AssertResults.ReportResult(ExpectedSize := SIZEOF(Expected),
                           ExpectedTypeClass := IBaseLibrary.TypeClass.TYPE_BYTE,
                           ExpectedValue := ADR(Expected),
                           ActualSize := SIZEOF(Actual),
                           ActualTypeClass := IBaseLibrary.TypeClass.TYPE_BYTE,
                           ActualValue := ADR(Actual),
                           Message := Message,
                           TestInstancePath := TestInstancePath,
                           AlreadyReported => AlreadyReported);

IF NOT AlreadyReported AND Expected <> Actual THEN
    SetTestFailed(AssertionType := E_AssertionType.Type_BYTE,
                  AssertionMessage := Message);

    AssertMessageFormatter.LogAssertFailure(Expected := CONCAT(
                                                       STR1 := '0x',
                                                       STR2 := BYTE_TO_HEXSTR(in := Expected,
                                                                                            iPrecision := 2,
                                                                                            bLoCase := FALSE)),
                                            Actual := CONCAT(
                                                       STR1 := '0x',
                                                       STR2 := BYTE_TO_HEXSTR(in := Actual,
                                                                                            iPrecision := 2,
                                                                                            bLoCase := FALSE)),
                                            Message := Message,
                                            TestInstancePath := TestInstancePath);
END_IF
END_METHOD

// Asserts that two DATEs are equal. If they are not, an assertion error is created.
METHOD PUBLIC AssertEquals_DATE
VAR_INPUT
    Expected : DATE; // DATE expected value
    Actual : DATE; // DATE actual value
    Message : T_MaxString; // The identifying message for the assertion error
END_VAR
VAR
    TestInstancePath : T_MaxString;
    AlreadyReported : BOOL;
END_VAR
IF GVL_TcUnit.IgnoreCurrentTest OR GVL_TcUnit.CurrentTestIsFinished THEN
    RETURN;
END_IF

TestInstancePath := AddTestNameToInstancePath(TestInstancePath := FindTestSuiteInstancePath());

AssertResults.ReportResult(ExpectedSize := SIZEOF(Expected),
                           ExpectedTypeClass := IBaseLibrary.TypeClass.TYPE_DATE,
                           ExpectedValue := ADR(Expected),
                           ActualSize := SIZEOF(Actual),
                           ActualTypeClass := IBaseLibrary.TypeClass.TYPE_DATE,
                           ActualValue := ADR(Actual),
                           Message := Message,
                           TestInstancePath := TestInstancePath,
                           AlreadyReported => AlreadyReported);

IF NOT AlreadyReported AND Expected <> Actual THEN
    SetTestFailed(AssertionType := E_AssertionType.Type_DATE,
                  AssertionMessage := Message);

    AssertMessageFormatter.LogAssertFailure(Expected := DATE_TO_STRING(Expected),
                                            Actual := DATE_TO_STRING(Actual),
                                            Message := Message,
                                            TestInstancePath := TestInstancePath);
END_IF
END_METHOD

// Asserts that two DATE_AND_TIMEs are equal. If they are not, an assertion error is created.
METHOD PUBLIC AssertEquals_DATE_AND_TIME
VAR_INPUT
    Expected : DATE_AND_TIME; // DATE_AND_TIME expected value
    Actual : DATE_AND_TIME; // DATE_AND_TIME actual value
    Message : T_MaxString; // The identifying message for the assertion error
END_VAR
VAR
    TestInstancePath : T_MaxString;
    AlreadyReported : BOOL;
END_VAR
IF GVL_TcUnit.IgnoreCurrentTest OR GVL_TcUnit.CurrentTestIsFinished THEN
    RETURN;
END_IF

TestInstancePath := AddTestNameToInstancePath(TestInstancePath := FindTestSuiteInstancePath());

AssertResults.ReportResult(ExpectedSize := SIZEOF(Expected),
                           ExpectedTypeClass := IBaseLibrary.TypeClass.TYPE_DATEANDTIME,
                           ExpectedValue := ADR(Expected),
                           ActualSize := SIZEOF(Actual),
                           ActualTypeClass := IBaseLibrary.TypeClass.TYPE_DATEANDTIME,
                           ActualValue := ADR(Actual),
                           Message := Message,
                           TestInstancePath := TestInstancePath,
                           AlreadyReported => AlreadyReported);

IF NOT AlreadyReported AND Expected <> Actual THEN
    SetTestFailed(AssertionType := E_AssertionType.Type_DATE_AND_TIME,
                  AssertionMessage := Message);

    AssertMessageFormatter.LogAssertFailure(Expected := DT_TO_STRING(Expected),
                                            Actual := DT_TO_STRING(Actual),
                                            Message := Message,
                                            TestInstancePath := TestInstancePath);
END_IF
END_METHOD

// Asserts that two DINTs are equal. If they are not, an assertion error is created.
METHOD PUBLIC AssertEquals_DINT
VAR_INPUT
    Expected : DINT; // DINT expected value
    Actual : DINT; // DINT actual value
    Message : T_MaxString; // The identifying message for the assertion error
END_VAR
VAR
    TestInstancePath : T_MaxString;
    AlreadyReported : BOOL;
END_VAR
IF GVL_TcUnit.IgnoreCurrentTest OR GVL_TcUnit.CurrentTestIsFinished THEN
    RETURN;
END_IF

TestInstancePath := AddTestNameToInstancePath(TestInstancePath := FindTestSuiteInstancePath());

AssertResults.ReportResult(ExpectedSize := SIZEOF(Expected),
                           ExpectedTypeClass := IBaseLibrary.TypeClass.TYPE_DINT,
                           ExpectedValue := ADR(Expected),
                           ActualSize := SIZEOF(Actual),
                           ActualTypeClass := IBaseLibrary.TypeClass.TYPE_DINT,
                           ActualValue := ADR(Actual),
                           Message := Message,
                           TestInstancePath := TestInstancePath,
                           AlreadyReported => AlreadyReported);

IF NOT AlreadyReported AND Expected <> Actual THEN
    SetTestFailed(AssertionType := E_AssertionType.Type_DINT,
                  AssertionMessage := Message);

    AssertMessageFormatter.LogAssertFailure(Expected := DINT_TO_STRING(Expected),
                                            Actual := DINT_TO_STRING(Actual),
                                            Message := Message,
                                            TestInstancePath := TestInstancePath);
END_IF
END_METHOD

// Asserts that two DWORDs are equal. If they are not, an assertion error is created.
METHOD PUBLIC AssertEquals_DWORD
VAR_INPUT
    Expected : DWORD; // DWORD expected value
    Actual : DWORD; // DWORD actual value
    Message : T_MaxString; // The identifying message for the assertion error
END_VAR
VAR
    TestInstancePath : T_MaxString;
    AlreadyReported : BOOL;
END_VAR
IF GVL_TcUnit.IgnoreCurrentTest OR GVL_TcUnit.CurrentTestIsFinished THEN
    RETURN;
END_IF

TestInstancePath := AddTestNameToInstancePath(TestInstancePath := FindTestSuiteInstancePath());

AssertResults.ReportResult(ExpectedSize := SIZEOF(Expected),
                           ExpectedTypeClass := IBaseLibrary.TypeClass.TYPE_DWORD,
                           ExpectedValue := ADR(Expected),
                           ActualSize := SIZEOF(Actual),
                           ActualTypeClass := IBaseLibrary.TypeClass.TYPE_DWORD,
                           ActualValue := ADR(Actual),
                           Message := Message,
                           TestInstancePath := TestInstancePath,
                           AlreadyReported => AlreadyReported);

IF NOT AlreadyReported AND Expected <> Actual THEN
    SetTestFailed(AssertionType := E_AssertionType.Type_DWORD,
                  AssertionMessage := Message);

    AssertMessageFormatter.LogAssertFailure(Expected := CONCAT(
                                                            STR1 := '0x',
                                                            STR2 := DWORD_TO_HEXSTR(in := Expected,
                                                                                                  iPrecision := 8,
                                                                                                  bLoCase := FALSE)),
                                            Actual := CONCAT(
                                                           STR1 := '0x',
                                                           STR2 := DWORD_TO_HEXSTR(in := Actual,
                                                                                                 iPrecision := 8,
                                                                                                 bLoCase := FALSE)),
                                            Message := Message,
                                            TestInstancePath := TestInstancePath);
END_IF
END_METHOD

// Asserts that two INTs are equal. If they are not, an assertion error is created.
METHOD PUBLIC AssertEquals_INT
VAR_INPUT
    Expected : INT; // INT expected value
    Actual : INT; // INT actual value
    Message : T_MaxString; // The identifying message for the assertion error
END_VAR
VAR
    TestInstancePath : T_MaxString;
    AlreadyReported : BOOL;
END_VAR
IF GVL_TcUnit.IgnoreCurrentTest OR GVL_TcUnit.CurrentTestIsFinished THEN
    RETURN;
END_IF

TestInstancePath := AddTestNameToInstancePath(TestInstancePath := FindTestSuiteInstancePath());

AssertResults.ReportResult(ExpectedSize := SIZEOF(Expected),
                           ExpectedTypeClass := IBaseLibrary.TypeClass.TYPE_INT,
                           ExpectedValue := ADR(Expected),
                           ActualSize := SIZEOF(Actual),
                           ActualTypeClass := IBaseLibrary.TypeClass.TYPE_INT,
                           ActualValue := ADR(Actual),
                           Message := Message,
                           TestInstancePath := TestInstancePath,
                           AlreadyReported => AlreadyReported);

IF NOT AlreadyReported AND Expected <> Actual THEN
    SetTestFailed(AssertionType := E_AssertionType.Type_INT,
                  AssertionMessage := Message);

    AssertMessageFormatter.LogAssertFailure(Expected := INT_TO_STRING(Expected),
                                            Actual := INT_TO_STRING(Actual),
                                            Message := Message,
                                            TestInstancePath := TestInstancePath);
END_IF
END_METHOD

// Asserts that two LINTs are equal. If they are not, an assertion error is created.
METHOD PUBLIC AssertEquals_LINT
VAR_INPUT
    Expected : LINT; // LINT expected value
    Actual : LINT; // LINT actual value
    Message : T_MaxString; // The identifying message for the assertion error
END_VAR
VAR
    TestInstancePath : T_MaxString;
    AlreadyReported : BOOL;
END_VAR
IF GVL_TcUnit.IgnoreCurrentTest OR GVL_TcUnit.CurrentTestIsFinished THEN
    RETURN;
END_IF

TestInstancePath := AddTestNameToInstancePath(TestInstancePath := FindTestSuiteInstancePath());

AssertResults.ReportResult(ExpectedSize := SIZEOF(Expected),
                           ExpectedTypeClass := IBaseLibrary.TypeClass.TYPE_LINT,
                           ExpectedValue := ADR(Expected),
                           ActualSize := SIZEOF(Actual),
                           ActualTypeClass := IBaseLibrary.TypeClass.TYPE_LINT,
                           ActualValue := ADR(Actual),
                           Message := Message,
                           TestInstancePath := TestInstancePath,
                           AlreadyReported => AlreadyReported);

IF NOT AlreadyReported AND Expected <> Actual THEN
    SetTestFailed(AssertionType := E_AssertionType.Type_LINT,
                  AssertionMessage := Message);

    AssertMessageFormatter.LogAssertFailure(Expected := LINT_TO_STRING(Expected),
                                            Actual := LINT_TO_STRING(Actual),
                                            Message := Message,
                                            TestInstancePath := TestInstancePath);
END_IF
END_METHOD

// Asserts that two LREALs are equal to within a positive delta. If they are not, an assertion error is created.
METHOD PUBLIC AssertEquals_LREAL
VAR_INPUT
    Expected : LREAL; // LREAL expected value
    Actual : LREAL; // LREAL actual value
    Delta : LREAL; // The maximum delta between the absolute value of expected and actual for which both numbers are still considered equal
    Message : T_MaxString; // The identifying message for the assertion error
END_VAR
VAR
    Equals : BOOL := TRUE;
    TestInstancePath : T_MaxString;
    AlreadyReported : BOOL;
END_VAR
IF GVL_TcUnit.IgnoreCurrentTest OR GVL_TcUnit.CurrentTestIsFinished THEN
    RETURN;
END_IF

TestInstancePath := AddTestNameToInstancePath(TestInstancePath := FindTestSuiteInstancePath());

AssertResults.ReportResult(ExpectedSize := SIZEOF(Expected),
                           ExpectedTypeClass := IBaseLibrary.TypeClass.TYPE_LREAL,
                           ExpectedValue := ADR(Expected),
                           ActualSize := SIZEOF(Actual),
                           ActualTypeClass := IBaseLibrary.TypeClass.TYPE_LREAL,
                           ActualValue := ADR(Actual),
                           Message := Message,
                           TestInstancePath := TestInstancePath,
                           AlreadyReported => AlreadyReported);

IF NOT AlreadyReported THEN
    IF LrealIsNaN (Delta) THEN
        Equals := FALSE;
        Message := CONCAT(STR1 := Message, STR2 := ', value of delta is NaN.');
    ELSIF (LrealIsNaN (Expected)
    OR     LrealIsNaN (Actual)) THEN
        Equals := FALSE;
        Message := CONCAT(STR1 := Message, STR2 := ', value of Expected or Actual is NaN.');
    ELSIF ABS(Expected - Actual) > Delta THEN
        Equals := FALSE;
    END_IF

    IF NOT Equals THEN
        SetTestFailed(AssertionType := E_AssertionType.Type_LREAL,
                      AssertionMessage := Message);

        AssertMessageFormatter.LogAssertFailure(Expected := LREAL_TO_STRING(Expected),
                                                Actual := LREAL_TO_STRING(Actual),
                                                Message := Message,
                                                TestInstancePath := TestInstancePath);
    END_IF
END_IF
END_METHOD

// Asserts that two LTIMEs are equal. If they are not, an assertion error is created.
METHOD PUBLIC AssertEquals_LTIME
VAR_INPUT
    Expected : LTIME; // LTIME expected value
    Actual : LTIME; // LTIME actual value
    Message : T_MaxString; // The identifying message for the assertion error
END_VAR
VAR
    TestInstancePath : T_MaxString;
    AlreadyReported : BOOL;
END_VAR
IF GVL_TcUnit.IgnoreCurrentTest OR GVL_TcUnit.CurrentTestIsFinished THEN
    RETURN;
END_IF

TestInstancePath := AddTestNameToInstancePath(TestInstancePath := FindTestSuiteInstancePath());

AssertResults.ReportResult(ExpectedSize := SIZEOF(Expected),
                           ExpectedTypeClass := IBaseLibrary.TypeClass.TYPE_LTIME,
                           ExpectedValue := ADR(Expected),
                           ActualSize := SIZEOF(Actual),
                           ActualTypeClass := IBaseLibrary.TypeClass.TYPE_LTIME,
                           ActualValue := ADR(Actual),
                           Message := Message,
                           TestInstancePath := TestInstancePath,
                           AlreadyReported => AlreadyReported);

IF NOT AlreadyReported AND Expected <> Actual THEN
    SetTestFailed(AssertionType := E_AssertionType.Type_LTIME,
                  AssertionMessage := Message);

    AssertMessageFormatter.LogAssertFailure(Expected := LTIME_TO_STRING(Expected),
                                            Actual := LTIME_TO_STRING(Actual),
                                            Message := Message,
                                            TestInstancePath := TestInstancePath);
END_IF
END_METHOD

// Asserts that two LWORDs are equal. If they are not, an assertion error is created.
METHOD PUBLIC AssertEquals_LWORD
VAR_INPUT
    Expected : LWORD; // LWORD expected value
    Actual : LWORD; // LWORD actual value
    Message : T_MaxString; // The identifying message for the assertion error
END_VAR
VAR
    TestInstancePath : T_MaxString;
    AlreadyReported : BOOL;
END_VAR
IF GVL_TcUnit.IgnoreCurrentTest OR GVL_TcUnit.CurrentTestIsFinished THEN
    RETURN;
END_IF

TestInstancePath := AddTestNameToInstancePath(TestInstancePath := FindTestSuiteInstancePath());

AssertResults.ReportResult(ExpectedSize := SIZEOF(Expected),
                           ExpectedTypeClass := IBaseLibrary.TypeClass.TYPE_LWORD,
                           ExpectedValue := ADR(Expected),
                           ActualSize := SIZEOF(Actual),
                           ActualTypeClass := IBaseLibrary.TypeClass.TYPE_LWORD,
                           ActualValue := ADR(Actual),
                           Message := Message,
                           TestInstancePath := TestInstancePath,
                           AlreadyReported => AlreadyReported);

IF NOT AlreadyReported AND Expected <> Actual THEN
    SetTestFailed(AssertionType := E_AssertionType.Type_LWORD,
                  AssertionMessage := Message);

    AssertMessageFormatter.LogAssertFailure(Expected := CONCAT(
                                                            STR1 := '0x',
                                                            STR2 := LWORD_TO_HEXSTR(in := Expected,
                                                                                                  iPrecision := 16,
                                                                                                  bLoCase := FALSE)),
                                            Actual := CONCAT(
                                                            STR1 := '0x',
                                                            STR2 := LWORD_TO_HEXSTR(in := Actual,
                                                                                                  iPrecision := 16,
                                                                                                  bLoCase := FALSE)),
                                            Message := Message,
                                            TestInstancePath := TestInstancePath);
END_IF
END_METHOD

// Asserts that two REALs are equal to within a positive delta. If they are not, an assertion error is created.
METHOD PUBLIC AssertEquals_REAL
VAR_INPUT
    Expected : REAL; // REAL expected value
    Actual : REAL; // REAL actual value
    Delta : REAL;  // The maximum delta between the absolute value of expected and actual for which both numbers are still considered equal
    Message : T_MaxString; // The identifying message for the assertion error
END_VAR
VAR
    Equals : BOOL := TRUE;
    TestInstancePath : T_MaxString;
    AlreadyReported : BOOL;
END_VAR
IF GVL_TcUnit.IgnoreCurrentTest OR GVL_TcUnit.CurrentTestIsFinished THEN
    RETURN;
END_IF

TestInstancePath := AddTestNameToInstancePath(TestInstancePath := FindTestSuiteInstancePath());

AssertResults.ReportResult(ExpectedSize := SIZEOF(Expected),
                           ExpectedTypeClass := IBaseLibrary.TypeClass.TYPE_REAL,
                           ExpectedValue := ADR(Expected),
                           ActualSize := SIZEOF(Actual),
                           ActualTypeClass := IBaseLibrary.TypeClass.TYPE_REAL,
                           ActualValue := ADR(Actual),
                           Message := Message,
                           TestInstancePath := TestInstancePath,
                           AlreadyReported => AlreadyReported);

IF NOT AlreadyReported THEN
    IF RealIsNaN (Delta) THEN
        Equals := FALSE;
        Message := CONCAT(STR1 := Message, STR2 := ', value of delta is NaN.');
    ELSIF (RealIsNaN (Expected)
    OR     RealIsNaN (Actual)) THEN
        Equals := FALSE;
        Message := CONCAT(STR1 := Message, STR2 := ', value of Expected or Actual is NaN.');
    ELSIF ABS(Expected - Actual) > Delta THEN
        Equals := FALSE;
    END_IF

    IF NOT Equals THEN
        SetTestFailed(AssertionType := E_AssertionType.Type_REAL,
                      AssertionMessage := Message);

        AssertMessageFormatter.LogAssertFailure(Expected := REAL_TO_STRING(Expected),
                                                Actual := REAL_TO_STRING(Actual),
                                                Message := Message,
                                                TestInstancePath := TestInstancePath);
    END_IF
END_IF
END_METHOD

// Asserts that two SINTs are equal. If they are not, an assertion error is created.
METHOD PUBLIC AssertEquals_SINT
VAR_INPUT
    Expected : SINT; // SINT expected value
    Actual : SINT; // SINT actual value
    Message : T_MaxString; // The identifying message for the assertion error
END_VAR
VAR
    TestInstancePath : T_MaxString;
    AlreadyReported : BOOL;
END_VAR
IF GVL_TcUnit.IgnoreCurrentTest OR GVL_TcUnit.CurrentTestIsFinished THEN
    RETURN;
END_IF

TestInstancePath := AddTestNameToInstancePath(TestInstancePath := FindTestSuiteInstancePath());

AssertResults.ReportResult(ExpectedSize := SIZEOF(Expected),
                           ExpectedTypeClass := IBaseLibrary.TypeClass.TYPE_SINT,
                           ExpectedValue := ADR(Expected),
                           ActualSize := SIZEOF(Actual),
                           ActualTypeClass := IBaseLibrary.TypeClass.TYPE_SINT,
                           ActualValue := ADR(Actual),
                           Message := Message,
                           TestInstancePath := TestInstancePath,
                           AlreadyReported => AlreadyReported);

IF NOT AlreadyReported AND Expected <> Actual THEN
    SetTestFailed(AssertionType := E_AssertionType.Type_SINT,
                  AssertionMessage := Message);

    AssertMessageFormatter.LogAssertFailure(Expected := SINT_TO_STRING(Expected),
                                            Actual := SINT_TO_STRING(Actual),
                                            Message := Message,
                                            TestInstancePath := TestInstancePath);
END_IF
END_METHOD

// Asserts that two STRINGs are equal. If they are not, an assertion error is created.
METHOD PUBLIC AssertEquals_STRING
VAR_INPUT
    Expected : T_MaxString; // STRING expected value
    Actual : T_MaxString; // STRING actual value
    Message : T_MaxString; // The identifying message for the assertion error
END_VAR
VAR
    TestInstancePath : T_MaxString;
    AlreadyReported : BOOL;
END_VAR
IF GVL_TcUnit.IgnoreCurrentTest OR GVL_TcUnit.CurrentTestIsFinished THEN
    RETURN;
END_IF

TestInstancePath := AddTestNameToInstancePath(TestInstancePath := FindTestSuiteInstancePath());

AssertResults.ReportResult(ExpectedSize := SIZEOF(Expected),
                           ExpectedTypeClass := IBaseLibrary.TypeClass.TYPE_STRING,
                           ExpectedValue := ADR(Expected),
                           ActualSize := SIZEOF(Actual),
                           ActualTypeClass := IBaseLibrary.TypeClass.TYPE_STRING,
                           ActualValue := ADR(Actual),
                           Message := Message,
                           TestInstancePath := TestInstancePath,
                           AlreadyReported => AlreadyReported);

IF NOT AlreadyReported AND (LEN(STR := Expected) <> LEN(STR := Actual) OR (Expected <> Actual)) THEN
    SetTestFailed(AssertionType := E_AssertionType.Type_STRING,
                  AssertionMessage := Message);

    AssertMessageFormatter.LogAssertFailure(Expected := Expected,
                                            Actual := Actual,
                                            Message := Message,
                                            TestInstancePath := TestInstancePath);
END_IF
END_METHOD

// Asserts that two TIMEs are equal. If they are not, an assertion error is created.
METHOD PUBLIC AssertEquals_TIME
VAR_INPUT
    Expected : TIME; // TIME expected value
    Actual : TIME; // TIME actual value
    Message : T_MaxString; // The identifying message for the assertion error
END_VAR
VAR
    TestInstancePath : T_MaxString;
    AlreadyReported : BOOL;
END_VAR
IF GVL_TcUnit.IgnoreCurrentTest OR GVL_TcUnit.CurrentTestIsFinished THEN
    RETURN;
END_IF

TestInstancePath := AddTestNameToInstancePath(TestInstancePath := FindTestSuiteInstancePath());

AssertResults.ReportResult(ExpectedSize := SIZEOF(Expected),
                           ExpectedTypeClass := IBaseLibrary.TypeClass.TYPE_TIME,
                           ExpectedValue := ADR(Expected),
                           ActualSize := SIZEOF(Actual),
                           ActualTypeClass := IBaseLibrary.TypeClass.TYPE_TIME,
                           ActualValue := ADR(Actual),
                           Message := Message,
                           TestInstancePath := TestInstancePath,
                           AlreadyReported => AlreadyReported);

IF NOT AlreadyReported AND Expected <> Actual THEN
    SetTestFailed(AssertionType := E_AssertionType.Type_TIME,
                  AssertionMessage := Message);

    AssertMessageFormatter.LogAssertFailure(Expected := TIME_TO_STRING(Expected),
                                            Actual := TIME_TO_STRING(Actual),
                                            Message := Message,
                                            TestInstancePath := TestInstancePath);
END_IF
END_METHOD

// Asserts that two TIME_OF_DAYs are equal. If they are not, an assertion error is created.
METHOD PUBLIC AssertEquals_TIME_OF_DAY
VAR_INPUT
    Expected : TIME_OF_DAY; // TIME_OF_DAY expected value
    Actual : TIME_OF_DAY; // TIME_OF_DAY actual value
    Message : T_MaxString; // The identifying message for the assertion error
END_VAR
VAR
    TestInstancePath : T_MaxString;
    AlreadyReported : BOOL;
END_VAR
IF GVL_TcUnit.IgnoreCurrentTest OR GVL_TcUnit.CurrentTestIsFinished THEN
    RETURN;
END_IF

TestInstancePath := AddTestNameToInstancePath(TestInstancePath := FindTestSuiteInstancePath());

AssertResults.ReportResult(ExpectedSize := SIZEOF(Expected),
                           ExpectedTypeClass := IBaseLibrary.TypeClass.TYPE_TIMEOFDAY,
                           ExpectedValue := ADR(Expected),
                           ActualSize := SIZEOF(Actual),
                           ActualTypeClass := IBaseLibrary.TypeClass.TYPE_TIMEOFDAY,
                           ActualValue := ADR(Actual),
                           Message := Message,
                           TestInstancePath := TestInstancePath,
                           AlreadyReported => AlreadyReported);

IF NOT AlreadyReported AND Expected <> Actual THEN
    SetTestFailed(AssertionType := E_AssertionType.Type_TIME_OF_DAY,
                  AssertionMessage := Message);

    AssertMessageFormatter.LogAssertFailure(Expected := TOD_TO_STRING(Expected),
                                            Actual := TOD_TO_STRING(Actual),
                                            Message := Message,
                                            TestInstancePath := TestInstancePath);
END_IF
END_METHOD

// Asserts that two UDINTs are equal. If they are not, an assertion error is created.
METHOD PUBLIC AssertEquals_UDINT
VAR_INPUT
    Expected : UDINT; // UDINT expected value
    Actual : UDINT; // UDINT actual value
    Message : T_MaxString; // The identifying message for the assertion error
END_VAR
VAR
    TestInstancePath : T_MaxString;
    AlreadyReported : BOOL;
END_VAR
IF GVL_TcUnit.IgnoreCurrentTest OR GVL_TcUnit.CurrentTestIsFinished THEN
    RETURN;
END_IF

TestInstancePath := AddTestNameToInstancePath(TestInstancePath := FindTestSuiteInstancePath());

AssertResults.ReportResult(ExpectedSize := SIZEOF(Expected),
                           ExpectedTypeClass := IBaseLibrary.TypeClass.TYPE_UDINT,
                           ExpectedValue := ADR(Expected),
                           ActualSize := SIZEOF(Actual),
                           ActualTypeClass := IBaseLibrary.TypeClass.TYPE_UDINT,
                           ActualValue := ADR(Actual),
                           Message := Message,
                           TestInstancePath := TestInstancePath,
                           AlreadyReported => AlreadyReported);

IF NOT AlreadyReported AND Expected <> Actual THEN
    SetTestFailed(AssertionType := E_AssertionType.Type_UDINT,
                  AssertionMessage := Message);

    AssertMessageFormatter.LogAssertFailure(Expected := UDINT_TO_STRING(Expected),
                                            Actual := UDINT_TO_STRING(Actual),
                                            Message := Message,
                                            TestInstancePath := TestInstancePath);
END_IF
END_METHOD

// Asserts that two UINTs are equal. If they are not, an assertion error is created.
METHOD PUBLIC AssertEquals_UINT
VAR_INPUT
    Expected : UINT; // UINT expected value
    Actual : UINT; // UINT actual value
    Message : T_MaxString; // The identifying message for the assertion error
END_VAR
VAR
    TestInstancePath : T_MaxString;
    AlreadyReported : BOOL;
END_VAR
IF GVL_TcUnit.IgnoreCurrentTest OR GVL_TcUnit.CurrentTestIsFinished THEN
    RETURN;
END_IF

TestInstancePath := AddTestNameToInstancePath(TestInstancePath := FindTestSuiteInstancePath());

AssertResults.ReportResult(ExpectedSize := SIZEOF(Expected),
                           ExpectedTypeClass := IBaseLibrary.TypeClass.TYPE_UINT,
                           ExpectedValue := ADR(Expected),
                           ActualSize := SIZEOF(Actual),
                           ActualTypeClass := IBaseLibrary.TypeClass.TYPE_UINT,
                           ActualValue := ADR(Actual),
                           Message := Message,
                           TestInstancePath := TestInstancePath,
                           AlreadyReported => AlreadyReported);

IF NOT AlreadyReported AND Expected <> Actual THEN
    SetTestFailed(AssertionType := E_AssertionType.Type_UINT,
                  AssertionMessage := Message);

    AssertMessageFormatter.LogAssertFailure(Expected := UINT_TO_STRING(Expected),
                                            Actual := UINT_TO_STRING(Actual),
                                            Message := Message,
                                            TestInstancePath := TestInstancePath);
END_IF
END_METHOD

// Asserts that two ULINTs are equal. If they are not, an assertion error is created.
METHOD PUBLIC AssertEquals_ULINT
VAR_INPUT
    Expected : ULINT; // ULINT expected value
    Actual : ULINT; // ULINT actual value
    Message : T_MaxString; // The identifying message for the assertion error
END_VAR
VAR
    TestInstancePath : T_MaxString;
    AlreadyReported : BOOL;
END_VAR
IF GVL_TcUnit.IgnoreCurrentTest OR GVL_TcUnit.CurrentTestIsFinished THEN
    RETURN;
END_IF

TestInstancePath := AddTestNameToInstancePath(TestInstancePath := FindTestSuiteInstancePath());

AssertResults.ReportResult(ExpectedSize := SIZEOF(Expected),
                           ExpectedTypeClass := IBaseLibrary.TypeClass.TYPE_ULINT,
                           ExpectedValue := ADR(Expected),
                           ActualSize := SIZEOF(Actual),
                           ActualTypeClass := IBaseLibrary.TypeClass.TYPE_ULINT,
                           ActualValue := ADR(Actual),
                           Message := Message,
                           TestInstancePath := TestInstancePath,
                           AlreadyReported => AlreadyReported);

IF NOT AlreadyReported AND Expected <> Actual THEN
    SetTestFailed(AssertionType := E_AssertionType.Type_ULINT,
                  AssertionMessage := Message);

    AssertMessageFormatter.LogAssertFailure(Expected := ULINT_TO_STRING(Expected),
                                            Actual := ULINT_TO_STRING(Actual),
                                            Message := Message,
                                            TestInstancePath := TestInstancePath);
END_IF
END_METHOD

// Asserts that two USINTs are equal. If they are not, an assertion error is created.
METHOD PUBLIC AssertEquals_USINT
VAR_INPUT
    Expected : USINT; // USINT expected value
    Actual : USINT; // USINT actual value
    Message : T_MaxString; // The identifying message for the assertion error
END_VAR
VAR
    AlreadyReported : BOOL;
    TestInstancePath : T_MaxString;
END_VAR
IF GVL_TcUnit.IgnoreCurrentTest OR GVL_TcUnit.CurrentTestIsFinished THEN
    RETURN;
END_IF

TestInstancePath := AddTestNameToInstancePath(TestInstancePath := FindTestSuiteInstancePath());

AssertResults.ReportResult(ExpectedSize := SIZEOF(Expected),
                           ExpectedTypeClass := IBaseLibrary.TypeClass.TYPE_USINT,
                           ExpectedValue := ADR(Expected),
                           ActualSize := SIZEOF(Actual),
                           ActualTypeClass := IBaseLibrary.TypeClass.TYPE_USINT,
                           ActualValue := ADR(Actual),
                           Message := Message,
                           TestInstancePath := TestInstancePath,
                           AlreadyReported => AlreadyReported);

IF NOT AlreadyReported AND Expected <> Actual THEN
    SetTestFailed(AssertionType := E_AssertionType.Type_USINT,
                  AssertionMessage := Message);

    AssertMessageFormatter.LogAssertFailure(Expected := USINT_TO_STRING(Expected),
                                            Actual := USINT_TO_STRING(Actual),
                                            Message := Message,
                                            TestInstancePath := TestInstancePath);
END_IF
END_METHOD

// Asserts that two WORDs are equal. If they are not, an assertion error is created.
METHOD PUBLIC AssertEquals_WORD
VAR_INPUT
    Expected : WORD; // WORD expected value
    Actual : WORD; // WORD actual value
    Message : T_MaxString; // The identifying message for the assertion error
END_VAR
VAR
    TestInstancePath : T_MaxString;
    AlreadyReported : BOOL;
END_VAR
IF GVL_TcUnit.IgnoreCurrentTest OR GVL_TcUnit.CurrentTestIsFinished THEN
    RETURN;
END_IF

TestInstancePath := AddTestNameToInstancePath(TestInstancePath := FindTestSuiteInstancePath());

AssertResults.ReportResult(ExpectedSize := SIZEOF(Expected),
                           ExpectedTypeClass := IBaseLibrary.TypeClass.TYPE_WORD,
                           ExpectedValue := ADR(Expected),
                           ActualSize := SIZEOF(Actual),
                           ActualTypeClass := IBaseLibrary.TypeClass.TYPE_WORD,
                           ActualValue := ADR(Actual),
                           Message := Message,
                           TestInstancePath := TestInstancePath,
                           AlreadyReported => AlreadyReported);

IF NOT AlreadyReported AND Expected <> Actual THEN
    SetTestFailed(AssertionType := E_AssertionType.Type_WORD,
                  AssertionMessage := Message);

    AssertMessageFormatter.LogAssertFailure(Expected := CONCAT(
                                                            STR1 := '0x',
                                                            STR2 := WORD_TO_HEXSTR(in := Expected,
                                                                                                 iPrecision := 4,
                                                                                                 bLoCase := FALSE)),
                                            Actual := CONCAT(
                                                            STR1 := '0x',
                                                            STR2 := WORD_TO_HEXSTR(in := Actual,
                                                                                                 iPrecision := 4,
                                                                                                 bLoCase := FALSE)),
                                            Message := Message,
                                            TestInstancePath := TestInstancePath);
END_IF
END_METHOD

// Asserts that two WSTRINGs are equal. If they are not, an assertion error is created.
METHOD PUBLIC AssertEquals_WSTRING
VAR_INPUT
    Expected : WSTRING(255); // WSTRING expected value
    Actual : WSTRING(255); // WSTRING actual value
    Message : T_MaxString; // The identifying message for the assertion error
END_VAR
VAR
    TestInstancePath : T_MaxString;
    AlreadyReported : BOOL;
END_VAR
IF GVL_TcUnit.IgnoreCurrentTest OR GVL_TcUnit.CurrentTestIsFinished THEN
    RETURN;
END_IF

TestInstancePath := AddTestNameToInstancePath(TestInstancePath := FindTestSuiteInstancePath());

AssertResults.ReportResult(ExpectedSize := SIZEOF(Expected),
                           ExpectedTypeClass := IBaseLibrary.TypeClass.TYPE_WSTRING,
                           ExpectedValue := ADR(Expected),
                           ActualSize := SIZEOF(Actual),
                           ActualTypeClass := IBaseLibrary.TypeClass.TYPE_WSTRING,
                           ActualValue := ADR(Actual),
                           Message := Message,
                           TestInstancePath := TestInstancePath,
                           AlreadyReported => AlreadyReported);

IF NOT AlreadyReported AND (WLEN(STR := Expected) <> WLEN(STR := Actual) OR (Expected <> Actual)) THEN
    SetTestFailed(AssertionType := E_AssertionType.Type_WSTRING,
                  AssertionMessage := Message);

    AssertMessageFormatter.LogAssertFailure(Expected := 'Not possible to print EXP unicode WSTRING value',
                                            Actual := 'Not possible to print ACT unicode WSTRING value',
                                            Message := Message,
                                            TestInstancePath := TestInstancePath);
END_IF
END_METHOD

// Asserts that a condition is false. If it is not, an assertion error is created.
METHOD PUBLIC AssertFalse
VAR_INPUT
    Condition : BOOL; // Condition to be checked
    Message : T_MaxString; // The identifying message for the assertion error
END_VAR
AssertEquals_BOOL(Expected := FALSE,
                  Actual := Condition,
                  Message := Message);
END_METHOD

// Asserts that a condition is true. If it is not, an assertion error is created.
METHOD PUBLIC AssertTrue
VAR_INPUT
    Condition : BOOL; // Condition to be checked
    Message : T_MaxString; // The identifying message for the assertion error
END_VAR
AssertEquals_BOOL(Expected := TRUE,
                  Actual := Condition,
                  Message := Message);
END_METHOD

METHOD INTERNAL CalculateAndSetNumberOfAssertsForTest
VAR_INPUT
    TestName : T_MaxString;
END_VAR
VAR
    TestInstancePath : T_MaxString;
    TotalNumberOfAsserts : UINT;
    NumberOfAsserts : UINT;
    NumberOfArrayAsserts : UINT;
    
    IteratorCounter : UINT;
END_VAR
TestInstancePath := AddTestNameToInstancePath(FindTestSuiteInstancePath());
NumberOfAsserts := AssertResults.GetNumberOfAssertsForTest(CompleteTestInstancePath := TestInstancePath);
NumberOfArrayAsserts := AssertArrayResults.GetNumberOfArrayAssertsForTest(CompleteTestInstancePath := TestInstancePath);
TotalNumberOfAsserts := NumberOfAsserts + NumberOfArrayAsserts;

IF TotalNumberOfAsserts > 0 THEN
    IF NumberOfTests > 0 THEN
        FOR IteratorCounter := 1 TO NumberOfTests BY 1 DO
            IF Tests[IteratorCounter].GetName() = TestName THEN
                Tests[IteratorCounter].SetNumberOfAssertions(NoOfAssertions := TotalNumberOfAsserts);
                RETURN;
            END_IF
        END_FOR
    END_IF
END_IF
END_METHOD

METHOD INTERNAL CalculateDuration
VAR_INPUT
    FinishedAt : LWORD; // CPU cycle counter with 100ns precision
END_VAR
IF Duration = 0.0 THEN
	Duration := LWORD_TO_LREAL(FinishedAt - StartedAt) * GVL_TcUnit.HundredNanosecondToSecond; // Seconds
END_IF
END_METHOD

METHOD FB_init : BOOL
VAR_INPUT
    bInitRetains : BOOL; // if TRUE, the retain variables are initialized (warm start / cold start)
    bInCopyCode : BOOL;  // if TRUE, the instance afterwards gets moved into the copy code (online change)
END_VAR
GVL_TcUnit.NumberOfInitializedTestSuites := GVL_TcUnit.NumberOfInitializedTestSuites + 1;
GVL_TcUnit.TestSuiteAddresses[GVL_TcUnit.NumberOfInitializedTestSuites] := THIS;
END_METHOD

// Searches for the instance path of the calling function block
METHOD PRIVATE FindTestSuiteInstancePath : T_MaxString
FindTestSuiteInstancePath := GetInstancePath();
END_METHOD

METHOD INTERNAL GetDuration : LREAL
GetDuration := Duration;
END_METHOD

METHOD INTERNAL GetHasStartedRunning : BOOL
GetHasStartedRunning := StartedAt > 0;
END_METHOD

METHOD INTERNAL GetInstancePath : T_MaxString
GetInstancePath := InstancePath;
END_METHOD

METHOD INTERNAL GetNumberOfFailedTests : UINT
VAR
    Counter : UINT;
    FailedTestsCount : UINT;
    NumberOfTestsToAnalyse : UINT(1..GVL_Param_TcUnit.MaxNumberOfTestsForEachTestSuite);
    NumberOfTestOverArrayLimit : UINT;
END_VAR
// Limit the test analyse to the max array limit of 'Tests[]'
NumberOfTestsToAnalyse := GetNumberOfTestsToAnalyse();
IF GetNumberOfTests() > NumberOfTestsToAnalyse THEN
    NumberOfTestOverArrayLimit := GetNumberOfTests()-NumberOfTestsToAnalyse;
END_IF

FOR Counter := 1 TO NumberOfTestsToAnalyse BY 1 DO
    IF Tests[Counter].IsFailed() THEN
        FailedTestsCount := FailedTestsCount + 1;
    END_IF
END_FOR

GetNumberOfFailedTests := FailedTestsCount + NumberOfTestOverArrayLimit;
END_METHOD

METHOD INTERNAL GetNumberOfSkippedTests : UINT
VAR
    Counter : UINT;
    SkippedTestsCount : UINT;
    NumberOfTestsToAnalyse : UINT(1..GVL_Param_TcUnit.MaxNumberOfTestsForEachTestSuite);
END_VAR
// Limit the test analyse to the max array limit of 'Tests[]'
NumberOfTestsToAnalyse := GetNumberOfTestsToAnalyse();

FOR Counter := 1 TO NumberOfTestsToAnalyse BY 1 DO
    IF Tests[Counter].IsSkipped() THEN
        SkippedTestsCount := SkippedTestsCount + 1;
    END_IF
END_FOR

GetNumberOfSkippedTests := SkippedTestsCount;
END_METHOD

METHOD INTERNAL GetNumberOfSuccessfulTests : UINT
GetNumberOfSuccessfulTests := GetNumberOfTests() - GetNumberOfFailedTests() - GetNumberOfSkippedTests();
END_METHOD

METHOD INTERNAL GetNumberOfTests : UINT
GetNumberOfTests := NumberOfTests;
END_METHOD

METHOD INTERNAL GetNumberOfTestsToAnalyse : UINT
GetNumberOfTestsToAnalyse := MIN(GetNumberOfTests(), GVL_Param_TcUnit.MaxNumberOfTestsForEachTestSuite);
END_METHOD

METHOD GetTestByName : REFERENCE TO FB_Test
VAR_INPUT
  TestName : T_MaxString;
END_VAR
VAR
  IteratorCounter : UINT;
  NumberOfTestsToAnalyse : UINT(1..GVL_Param_TcUnit.MaxNumberOfTestSuites);
END_VAR
NumberOfTestsToAnalyse := GetNumberOfTestsToAnalyse();
FOR IteratorCounter := 1 TO NumberOfTestsToAnalyse BY 1 DO
  IF Tests[IteratorCounter].GetName() = TestName THEN
    GetTestByName REF= Tests[IteratorCounter];
    RETURN;
	END_IF
END_FOR
END_METHOD

// This method returns the test at the n'th position, ranging from 1.. NumberOfTests
METHOD INTERNAL GetTestByPosition : FB_Test
VAR_INPUT
    Position : UINT(1..GVL_Param_TcUnit.MaxNumberOfTestsForEachTestSuite);
END_VAR
GetTestByPosition := Tests[Position];
END_METHOD

METHOD INTERNAL GetTestOrderNumber : UINT(0..GVL_Param_TcUnit.MaxNumberOfTestsForEachTestSuite);
VAR_INPUT
    TestName : T_MaxString;
END_VAR
VAR
    IteratorCounter : UINT;
    NumberOfTestsToAnalyse : UINT(1..GVL_Param_TcUnit.MaxNumberOfTestsForEachTestSuite);
END_VAR
// Limit the test analyse to the max array limit of 'Tests[]'
NumberOfTestsToAnalyse := GetNumberOfTestsToAnalyse();

FOR IteratorCounter := 1 TO NumberOfTestsToAnalyse BY 1 DO
    IF Tests[IteratorCounter].GetName() = TestName THEN
        GetTestOrderNumber := Tests[IteratorCounter].GetTestOrder();
        RETURN;
    END_IF
END_FOR
END_METHOD

METHOD INTERNAL IsTestFinished : BOOL
VAR_INPUT
    TestName : T_MaxString;
END_VAR
VAR
    IteratorCounter : UINT;
    NumberOfTestsToAnalyse : UINT(0..GVL_Param_TcUnit.MaxNumberOfTestsForEachTestSuite);
END_VAR
// Limit the test analyse to the max array limit of 'Tests[]'
NumberOfTestsToAnalyse := GetNumberOfTestsToAnalyse();

IsTestFinished := FALSE;
FOR IteratorCounter := 1 TO NumberOfTestsToAnalyse BY 1 DO
    IF Tests[IteratorCounter].GetName() = TestName THEN
        IsTestFinished := Tests[IteratorCounter].IsFinished();
        RETURN;
    END_IF
END_FOR
END_METHOD

METHOD INTERNAL SetStartedAtIfNotSet
VAR_INPUT
    Timestamp : LWORD; // CPU cycle counter with 100ns precision
END_VAR
IF StartedAt = 0 THEN
    StartedAt := Timestamp;
END_IF
END_METHOD

METHOD INTERNAL SetStartedAtTimeBasedOnCpuCounter
StartedAt := F_GetCpuCounterAs64bit(GVL_TcUnit.GetCpuCounter);
END_METHOD

METHOD PRIVATE SetTestFailed
VAR_INPUT
    AssertionType : E_AssertionType;
    AssertionMessage : T_MaxString;
END_VAR
VAR
    IteratorCounter : UINT;
    NumberOfTestsToAnalyse : UINT(0..GVL_Param_TcUnit.MaxNumberOfTestsForEachTestSuite);
END_VAR
// Limit the test analyse to the max array limit of 'Tests[]'
NumberOfTestsToAnalyse := GetNumberOfTestsToAnalyse();

FOR IteratorCounter := 1 TO NumberOfTestsToAnalyse BY 1 DO
    IF Tests[IteratorCounter].GetName() = GVL_TcUnit.CurrentTestNameBeingCalled THEN
        Tests[IteratorCounter].SetFailed();
        Tests[IteratorCounter].SetAssertionType(AssertType := AssertionType);
        Tests[IteratorCounter].SetAssertionMessage(AssertMessage := AssertionMessage);
    END_IF
END_FOR
END_METHOD

(* Marks the test as finished in this testsuite.
   Returns TRUE if test was found, and FALSE if a test with this name was not found in this testsuite *)
METHOD INTERNAL SetTestFinished : BOOL;
VAR_INPUT
    TestName : T_MaxString;
    FinishedAt : LWORD;
END_VAR
VAR
    IteratorCounter : UINT;
    NumberOfTestsToAnalyse : UINT(0..GVL_Param_TcUnit.MaxNumberOfTestsForEachTestSuite);
END_VAR
// Limit the test analyse to the max array limit of 'Tests[]'
NumberOfTestsToAnalyse := GetNumberOfTestsToAnalyse();
FOR IteratorCounter := 1 TO NumberOfTestsToAnalyse BY 1 DO
    IF Tests[IteratorCounter].GetName() = TestName THEN
		IF NOT Tests[IteratorCounter].IsFinished() THEN
        	Tests[IteratorCounter].SetFinishedAndDuration(FinishedAt := FinishedAt);
		END_IF
		SetTestFinished := TRUE;
        RETURN;
    END_IF
END_FOR
SetTestFinished := FALSE;
END_METHOD

END_FUNCTION_BLOCK

// ---- POUs/FB_AssertResultStatic.TcPOU
(*
    This function block is responsible for keeping track of which asserts that have been made. The reason we need to
    keep track of these is because if the user does the same assert twice (because of running a test suite over several
    PLC-cycles) we want to know it so we don't print several times (if the assert fails).
    An instance of an assert is keyed/identified with the following parameters as key:
    - Value of expected
    - Value of actual
    - Message (string)
    - Test instance path (string)
*)
FUNCTION_BLOCK FB_AssertResultStatic
VAR
    // The total number of instances of each of the "AssertResults"
    AssertResults : ARRAY[1..GVL_Param_TcUnit.MaxNumberOfAssertsForEachTestSuite] OF ST_AssertResult;

    // The total number of unique asserts
    TotalAsserts : UINT := 0;

    // Function block to get the current task cycle
    GetCurrentTaskIndex : GETCURTASKINDEX;

    // The total number of instances of each of the "AssertResults"
    AssertResultInstances : ARRAY[1..GVL_Param_TcUnit.MaxNumberOfAssertsForEachTestSuite] OF ST_AssertResultInstances;

    // The last PLC cycle count
    CycleCount : UDINT;

    // Only run first cycle
    FirstCycleExecuted : BOOL;
END_VAR

METHOD PRIVATE AddAssertResult
VAR_INPUT
    ExpectedSize : UDINT;
    ExpectedTypeClass : IBaseLibrary.TypeClass;
    ExpectedValue : POINTER TO BYTE;
    ActualSize : UDINT;
    ActualTypeClass : IBaseLibrary.TypeClass;
    ActualValue : POINTER TO BYTE;
    Message : T_MaxString;
    TestInstancePath : T_MaxString;
END_VAR
VAR_INST
	AssertResultOverflow : BOOL := FALSE;
END_VAR
VAR
    sErrorString : T_MaxString;
END_VAR
IF TotalAsserts < GVL_Param_TcUnit.MaxNumberOfAssertsForEachTestSuite THEN
    TotalAsserts := TotalAsserts + 1;
    AssertResults[TotalAsserts].Expected := F_AnyToUnionValue(AnySize := ExpectedSize, AnyTypeClass := ExpectedTypeClass, AnyValue := ExpectedValue);
    AssertResults[TotalAsserts].Actual := F_AnyToUnionValue(AnySize := ActualSize, AnyTypeClass := ActualTypeClass, AnyValue := ActualValue);
    AssertResults[TotalAsserts].Message := Message;
    AssertResults[TotalAsserts].TestInstancePath := TestInstancePath;
ELSE
    IF NOT AssertResultOverflow THEN
        sErrorString := CONCAT(STR1 := F_GetTestSuiteNameFromTestInstancePath(TestInstancePath := TestInstancePath),
                               STR2 := '. Max number of assertions exceeded. Check parameter MaxNumberOfAssertsForEachTestSuite.');
		GVL_TcUnit.AdsMessageQueue.WriteLog(msgCtrlMask := ADSLOG_MSGTYPE_ERROR,
											msgFmtStr := sErrorString,
											strArg := '');
		AssertResultOverflow := TRUE;
	END_IF
END_IF
END_METHOD

METHOD PRIVATE CopyDetectionCountAndResetDetectionCountInThisCycle
VAR
    IteratorCounter : UINT;
END_VAR
FOR IteratorCounter := 1 TO GVL_Param_TcUnit.MaxNumberOfAssertsForEachTestSuite BY 1 DO
    AssertResultInstances[IteratorCounter].DetectionCount := AssertResultInstances[IteratorCounter].DetectionCountThisCycle;
    AssertResultInstances[IteratorCounter].DetectionCountThisCycle := 0;
END_FOR
END_METHOD

METHOD PRIVATE CreateAssertResultInstance
VAR_INPUT
    ExpectedSize : UDINT;
    ExpectedTypeClass : IBaseLibrary.TypeClass;
    ExpectedValue : POINTER TO BYTE;
    ActualSize : UDINT;
    ActualTypeClass : IBaseLibrary.TypeClass;
    ActualValue : POINTER TO BYTE;
    Message : T_MaxString;
    TestInstancePath : T_MaxString;
END_VAR
VAR
    IteratorCounter : UINT;
END_VAR
FOR IteratorCounter := 1 TO GVL_Param_TcUnit.MaxNumberOfAssertsForEachTestSuite BY 1 DO
    IF AssertResultInstances[IteratorCounter].DetectionCount = 0 AND
        AssertResultInstances[IteratorCounter].DetectionCountThisCycle = 0 THEN // Find first free spot
        AssertResultInstances[IteratorCounter].AssertResult.Expected := F_AnyToUnionValue(AnySize := ExpectedSize, AnyTypeClass := ExpectedTypeClass, AnyValue := ExpectedValue);
        AssertResultInstances[IteratorCounter].AssertResult.Actual := F_AnyToUnionValue(AnySize := ActualSize, AnyTypeClass := ActualTypeClass, AnyValue := ActualValue);
        AssertResultInstances[IteratorCounter].AssertResult.Message := Message;
        AssertResultInstances[IteratorCounter].AssertResult.TestInstancePath := TestInstancePath;
        AssertResultInstances[IteratorCounter].DetectionCountThisCycle := 1;
        EXIT;
    END_IF
END_FOR
END_METHOD

METHOD PRIVATE GetDetectionCount : UINT
VAR_INPUT
    ExpectedSize : UDINT;
    ExpectedTypeClass : IBaseLibrary.TypeClass;
    ExpectedValue : POINTER TO BYTE;
    ActualSize : UDINT;
    ActualTypeClass : IBaseLibrary.TypeClass;
    ActualValue : POINTER TO BYTE;
    Message : T_MaxString;
    TestInstancePath : T_MaxString;
END_VAR
VAR
    IteratorCounter : UINT;
END_VAR
FOR IteratorCounter := 1 TO GVL_Param_TcUnit.MaxNumberOfAssertsForEachTestSuite BY 1 DO
    IF F_IsAnyEqualToUnionValue(ExpectedOrActual := AssertResultInstances[IteratorCounter].AssertResult.Expected,
                                ExpectedOrActualSize := ExpectedSize,
                                ExpectedOrActualTypeClass := ExpectedTypeClass,
                                ExpectedOrActualValue := ExpectedValue) AND
       F_IsAnyEqualToUnionValue(ExpectedOrActual := AssertResultInstances[IteratorCounter].AssertResult.Actual,
                                ExpectedOrActualSize := ActualSize,
                                ExpectedOrActualTypeClass := ActualTypeClass,
                                ExpectedOrActualValue := ActualValue) AND
        AssertResultInstances[IteratorCounter].AssertResult.Message = Message AND
        AssertResultInstances[IteratorCounter].AssertResult.TestInstancePath = TestInstancePath THEN
        GetDetectionCount := AssertResultInstances[IteratorCounter].DetectionCount;
    END_IF
END_FOR
END_METHOD

METHOD PRIVATE GetDetectionCountThisCycle : UINT
VAR_INPUT
    ExpectedSize : UDINT;
    ExpectedTypeClass : IBaseLibrary.TypeClass;
    ExpectedValue : POINTER TO BYTE;
    ActualSize : UDINT;
    ActualTypeClass : IBaseLibrary.TypeClass;
    ActualValue : POINTER TO BYTE;
    Message : T_MaxString;
    TestInstancePath : T_MaxString;
END_VAR
VAR
    IteratorCounter : UINT;
END_VAR
FOR IteratorCounter := 1 TO GVL_Param_TcUnit.MaxNumberOfAssertsForEachTestSuite BY 1 DO
    IF F_IsAnyEqualToUnionValue(ExpectedOrActual := AssertResultInstances[IteratorCounter].AssertResult.Expected,
                                ExpectedOrActualSize := ExpectedSize,
                                ExpectedOrActualTypeClass := ExpectedTypeClass,
                                ExpectedOrActualValue := ExpectedValue) AND
       F_IsAnyEqualToUnionValue(ExpectedOrActual := AssertResultInstances[IteratorCounter].AssertResult.Actual,
                                ExpectedOrActualSize := ActualSize,
                                ExpectedOrActualTypeClass := ActualTypeClass,
                                ExpectedOrActualValue := ActualValue) AND
        AssertResultInstances[IteratorCounter].AssertResult.Message = Message AND
        AssertResultInstances[IteratorCounter].AssertResult.Message = TestInstancePath THEN
        GetDetectionCountThisCycle := AssertResultInstances[IteratorCounter].DetectionCountThisCycle;
    END_IF
END_FOR
END_METHOD

METHOD INTERNAL GetNumberOfAssertsForTest : UINT
VAR_INPUT
    CompleteTestInstancePath : T_MaxString;
END_VAR
VAR
    Counter : UINT;
    NumberOfAsserts : UINT := 0;
END_VAR
IF TotalAsserts > 0 THEN
    FOR Counter := 1 TO TotalAsserts BY 1 DO
        IF AssertResults[Counter].TestInstancePath = CompleteTestInstancePath THEN
            NumberOfAsserts := NumberOfAsserts + 1;
        END_IF
    END_FOR
END_IF

GetNumberOfAssertsForTest := NumberOfAsserts;
END_METHOD

(*
    This method is called in every assert and returns whether this particular assert has already been called.
    The reason one would like to know whether this assert has already been reported or not is to not report it several
    times to any logging service. Because a test-suite can consist of several tests, and certain tests can require the
    test to run over several cycles it means that certain asserts could be called several times and thus we need to
    keep track of which asserts we've already reported. The user of the framework should not need to care for any of
    this and he/she should be able to call the asserts in any way they find suitable.

    To know what assert this is we need to check for the total combination of:
    - Test message
    - Test instance path
    - Expected value
    - Actual value
    Theoretically we can have a situation where a test has three different asserts, each and one with the same test
    message/test instance path/actual value/expected value but called within the same or different cycles. In order for
    us to handle all situations we need a simple algorithm that works according to:
    - Keep track of how many instances the combination of test message/test instance path/expected value/actual value
      we have. So for example, if we have called Assert(Exp := 5, Act := 5, 'Hello there', 'PRG.InstanceTestSuite.Test')
      two times in one cycle, we have two instances of that combination. This is done according to:
    - Iterate all existing reports.
      - If we have a new PLC-cycle, set the current detection-count to zero.
      - If new report does not match in any of the above fields, create it (together with current PLC-cycle).
        Also store the information that we have one instance of this combination and +1 on the detection-count.
      - If new report matches in all of the above, +1 in the detection-count. If this detection-count is larger than
        the stored detection-count for this combination, create a new report and add +1 to the storage of
        the detection-count.
*)
METHOD INTERNAL ReportResult
VAR_INPUT
    ExpectedSize : UDINT;
    ExpectedTypeClass : IBaseLibrary.TypeClass;
    ExpectedValue : POINTER TO BYTE;
    ActualSize : UDINT;
    ActualTypeClass : IBaseLibrary.TypeClass;
    ActualValue : POINTER TO BYTE;
    Message : T_MaxString;
    TestInstancePath : T_MaxString;
END_VAR
VAR_OUTPUT
    AlreadyReported : BOOL := FALSE;
END_VAR
VAR
    LocationIndex : UINT;
    DataTypesNotEquals : BOOL;
    DataSizeNotEquals : BOOL;
    DataContentNotEquals : BOOL;
    CurrentCycleCount : UDINT;
    IteratorCounter : UINT;
    DetectionCountTemp : UINT := 0;
    FoundOne : BOOL;
    AdditionalIdenticalAssert : BOOL;
END_VAR
IF NOT FirstCycleExecuted THEN
    GetCurrentTaskIndex();
    FirstCycleExecuted := TRUE;
END_IF

CurrentCycleCount := TwinCAT_SystemInfoVarList._TaskInfo[GetCurrentTaskIndex.index].CycleCount;
(* Is current cycle the same as the last call to this method?
   If not, reset the detection count *)
IF CurrentCycleCount <> CycleCount THEN
    CopyDetectionCountAndResetDetectionCountInThisCycle();
END_IF

FOR IteratorCounter := 1 TO TotalAsserts BY 1 DO
      IF F_IsAnyEqualToUnionValue(ExpectedOrActual := AssertResultInstances[IteratorCounter].AssertResult.Expected,
                                  ExpectedOrActualSize := ExpectedSize,
                                  ExpectedOrActualTypeClass := ExpectedTypeClass,
                                  ExpectedOrActualValue := ExpectedValue) AND
         F_IsAnyEqualToUnionValue(ExpectedOrActual := AssertResultInstances[IteratorCounter].AssertResult.Actual,
                                  ExpectedOrActualSize := ActualSize,
                                  ExpectedOrActualTypeClass := ActualTypeClass,
                                  ExpectedOrActualValue := ActualValue) AND
        AssertResultInstances[IteratorCounter].AssertResult.Message = Message AND
        AssertResultInstances[IteratorCounter].AssertResult.TestInstancePath = TestInstancePath THEN
            AssertResultInstances[IteratorCounter].DetectionCountThisCycle :=
                AssertResultInstances[IteratorCounter].DetectionCountThisCycle + 1;
            FoundOne := TRUE;
        IF AssertResultInstances[IteratorCounter].DetectionCountThisCycle >
            AssertResultInstances[IteratorCounter].DetectionCount THEN // This assert is new
            AdditionalIdenticalAssert := TRUE;
        END_IF
        EXIT;
    END_IF
END_FOR

// If not found anything, create the first
IF NOT FoundOne THEN
    // No existing match found, create a new entry
    AddAssertResult(ExpectedSize := ExpectedSize,
                    ExpectedTypeClass := ExpectedTypeClass,
                    ExpectedValue := ExpectedValue,
                    ActualSize := ActualSize,
                    ActualTypeClass := ActualTypeClass,
                    ActualValue := ActualValue,
                    Message := Message, TestInstancePath := TestInstancePath);

    CreateAssertResultInstance(ExpectedSize := ExpectedSize,
                               ExpectedTypeClass := ExpectedTypeClass,
                               ExpectedValue := ExpectedValue,
                               ActualSize := ActualSize,
                               ActualTypeClass := ActualTypeClass,
                               ActualValue := ActualValue,
                               Message := Message, TestInstancePath := TestInstancePath);
// An additional instance of this assert needs to be created
ELSIF AdditionalIdenticalAssert THEN
    AddAssertResult(ExpectedSize := ExpectedSize,
                    ExpectedTypeClass := ExpectedTypeClass,
                    ExpectedValue := ExpectedValue,
                    ActualSize := ActualSize,
                    ActualTypeClass := ActualTypeClass,
                    ActualValue := ActualValue,
                    Message := Message, TestInstancePath := TestInstancePath);
// In all other cases, this assert has already been reported, we don't need to do anything
ELSE
    AlreadyReported := TRUE;
END_IF

// Update the cycle count
CycleCount := TwinCAT_SystemInfoVarList._TaskInfo[GetCurrentTaskIndex.index].CycleCount;
END_METHOD

END_FUNCTION_BLOCK

// ---- POUs/Functions/F_AnyToUnionValue.TcPOU
FUNCTION F_AnyToUnionValue : U_ExpectedOrActual
VAR_INPUT
    AnySize : UDINT;
    AnyTypeClass : IBaseLibrary.TypeClass;
    AnyValue : POINTER TO BYTE;
END_VAR

CASE AnyTypeClass OF
    IBaseLibrary.TypeClass.TYPE_BOOL :
        MEMCPY(destaddr := ADR(F_AnyToUnionValue.boolExpectedOrActual),
               srcAddr := AnyValue,
               n := AnySize);

    IBaseLibrary.TypeClass.TYPE_BIT :
        {warning disable C0355}
        MEMCPY(destaddr := ADR(F_AnyToUnionValue.bitExpectedOrActual),
               srcAddr := AnyValue,
               n := AnySize);
        {warning enable C0355}

    IBaseLibrary.TypeClass.TYPE_BYTE :
        MEMCPY(destaddr := ADR(F_AnyToUnionValue.byteExpectedOrActual),
               srcAddr := AnyValue,
               n := AnySize);

    IBaseLibrary.TypeClass.TYPE_WORD :
        MEMCPY(destaddr := ADR(F_AnyToUnionValue.wordExpectedOrActual),
               srcAddr := AnyValue,
               n := AnySize);

    IBaseLibrary.TypeClass.TYPE_DWORD :
        MEMCPY(destaddr := ADR(F_AnyToUnionValue.dwordExpectedOrActual),
               srcAddr := AnyValue,
               n := AnySize);

    IBaseLibrary.TypeClass.TYPE_LWORD :
        MEMCPY(destaddr := ADR(F_AnyToUnionValue.lwordExpectedOrActual),
               srcAddr := AnyValue,
               n := AnySize);

    IBaseLibrary.TypeClass.TYPE_SINT :
        MEMCPY(destaddr := ADR(F_AnyToUnionValue.sintExpectedOrActual),
               srcAddr := AnyValue,
               n := AnySize);

    IBaseLibrary.TypeClass.TYPE_INT :
        MEMCPY(destaddr := ADR(F_AnyToUnionValue.intExpectedOrActual),
               srcAddr := AnyValue,
               n := AnySize);

    IBaseLibrary.TypeClass.TYPE_DINT :
        MEMCPY(destaddr := ADR(F_AnyToUnionValue.dintExpectedOrActual),
               srcAddr := AnyValue,
               n := AnySize);

    IBaseLibrary.TypeClass.TYPE_LINT :
        MEMCPY(destaddr := ADR(F_AnyToUnionValue.lintExpectedOrActual),
               srcAddr := AnyValue,
               n := AnySize);

    IBaseLibrary.TypeClass.TYPE_USINT :
        MEMCPY(destaddr := ADR(F_AnyToUnionValue.usintExpectedOrActual),
               srcAddr := AnyValue,
               n := AnySize);

    IBaseLibrary.TypeClass.TYPE_UINT :
        MEMCPY(destaddr := ADR(F_AnyToUnionValue.uintExpectedOrActual),
               srcAddr := AnyValue,
               n := AnySize);

    IBaseLibrary.TypeClass.TYPE_UDINT :
        MEMCPY(destaddr := ADR(F_AnyToUnionValue.udintExpectedOrActual),
               srcAddr := AnyValue,
               n := AnySize);

    IBaseLibrary.TypeClass.TYPE_ULINT :
        MEMCPY(destaddr := ADR(F_AnyToUnionValue.ulintExpectedOrActual),
               srcAddr := AnyValue,
               n := AnySize);

    IBaseLibrary.TypeClass.TYPE_REAL :
        MEMCPY(destaddr := ADR(F_AnyToUnionValue.realExpectedOrActual),
               srcAddr := AnyValue,
               n := AnySize);

    IBaseLibrary.TypeClass.TYPE_LREAL :
        MEMCPY(destaddr := ADR(F_AnyToUnionValue.lrealExpectedOrActual),
               srcAddr := AnyValue,
               n := AnySize);

    IBaseLibrary.TypeClass.TYPE_STRING :
        MEMCPY(destaddr := ADR(F_AnyToUnionValue.stringExpectedOrActual),
               srcAddr := AnyValue,
               n := AnySize);

    IBaseLibrary.TypeClass.TYPE_WSTRING :
        MEMCPY(destaddr := ADR(F_AnyToUnionValue.wstringExpectedOrActual),
               srcAddr := AnyValue,
               n := AnySize);

    IBaseLibrary.TypeClass.TYPE_TIME :
        MEMCPY(destaddr := ADR(F_AnyToUnionValue.timeExpectedOrActual),
               srcAddr := AnyValue,
               n := AnySize);

    IBaseLibrary.TypeClass.TYPE_DATE :
        MEMCPY(destaddr := ADR(F_AnyToUnionValue.dateExpectedOrActual),
               srcAddr := AnyValue,
               n := AnySize);

    IBaseLibrary.TypeClass.TYPE_DATEANDTIME :
        MEMCPY(destaddr := ADR(F_AnyToUnionValue.dateandtimeExpectedOrActual),
               srcAddr := AnyValue,
               n := AnySize);

    IBaseLibrary.TypeClass.TYPE_TIMEOFDAY :
        MEMCPY(destaddr := ADR(F_AnyToUnionValue.timeofdayExpectedOrActual),
               srcAddr := AnyValue,
               n := AnySize);

    IBaseLibrary.TypeClass.TYPE_POINTER :
        // None

    IBaseLibrary.TypeClass.TYPE_REFERENCE :
        // None

    IBaseLibrary.TypeClass.TYPE_SUBRANGE :
        // None

    IBaseLibrary.TypeClass.TYPE_ENUM :
        // None

    IBaseLibrary.TypeClass.TYPE_ARRAY :
        // None

    IBaseLibrary.TypeClass.TYPE_PARAMS :
        // None

    IBaseLibrary.TypeClass.TYPE_USERDEF :
        // None

    IBaseLibrary.TypeClass.TYPE_NONE :
        // None

    IBaseLibrary.TypeClass.TYPE_ANY :
        // None

    IBaseLibrary.TypeClass.TYPE_ANYBIT :
        // None

    IBaseLibrary.TypeClass.TYPE_ANYDATE :
        // None

    IBaseLibrary.TypeClass.TYPE_ANYINT :
        // None

    IBaseLibrary.TypeClass.TYPE_ANYNUM :
        // None

    IBaseLibrary.TypeClass.TYPE_ANYREAL :
        // None

    IBaseLibrary.TypeClass.TYPE_LAZY :
        // None

    IBaseLibrary.TypeClass.TYPE_LTIME :
        MEMCPY(destaddr := ADR(F_AnyToUnionValue.ltimeExpectedOrActual),
               srcAddr := AnyValue,
               n := AnySize);

    IBaseLibrary.TypeClass.TYPE_BITCONST :
        // None

    IBaseLibrary.TypeClass.TYPE_INTERFACE :
        // None

    ELSE
        // None
END_CASE

END_FUNCTION

// ---- POUs/Functions/F_GetTestSuiteNameFromTestInstancePath.TcPOU
FUNCTION F_GetTestSuiteNameFromTestInstancePath : T_MaxString
VAR_INPUT
    TestInstancePath : T_MaxString;
END_VAR
VAR
    TestSuiteName : T_MaxString;
    FindPosition : INT;
END_VAR

TestSuiteName := F_RemoveInstancePathAndProjectNameFromTestInstancePath(TestInstancePath := TestInstancePath);
// Remove everything except the test suite name
FindPosition := FIND(STR1 := TestSuiteName, '.');
TestSuiteName := RIGHT(STR := TestSuiteName, SIZE := LEN(STR := TestSuiteName) - FindPosition);
F_GetTestSuiteNameFromTestInstancePath := TestSuiteName;

END_FUNCTION

// ---- POUs/Functions/F_IsAnyEqualToUnionValue.TcPOU
FUNCTION F_IsAnyEqualToUnionValue : BOOL
VAR_INPUT
    ExpectedOrActual : U_ExpectedOrActual;
    ExpectedOrActualSize : UDINT;
    ExpectedOrActualTypeClass : IBaseLibrary.TypeClass;
    ExpectedOrActualValue : POINTER TO BYTE;
END_VAR
VAR
    AnyExpectedOrActual : U_ExpectedOrActual;
END_VAR

AnyExpectedOrActual := F_AnyToUnionValue(AnySize := ExpectedOrActualSize,
                                         AnyTypeClass := ExpectedOrActualTypeClass,
                                         AnyValue := ExpectedOrActualValue);

CASE ExpectedOrActualTypeClass OF

    IBaseLibrary.TypeClass.TYPE_BOOL :
        F_IsAnyEqualToUnionValue := ExpectedOrActual.boolExpectedOrActual = AnyExpectedOrActual.boolExpectedOrActual;

    IBaseLibrary.TypeClass.TYPE_BIT :
        F_IsAnyEqualToUnionValue := ExpectedOrActual.bitExpectedOrActual = AnyExpectedOrActual.bitExpectedOrActual;

    IBaseLibrary.TypeClass.TYPE_BYTE :
        F_IsAnyEqualToUnionValue := ExpectedOrActual.byteExpectedOrActual = AnyExpectedOrActual.byteExpectedOrActual;

    IBaseLibrary.TypeClass.TYPE_WORD :
        F_IsAnyEqualToUnionValue := ExpectedOrActual.wordExpectedOrActual = AnyExpectedOrActual.wordExpectedOrActual;

    IBaseLibrary.TypeClass.TYPE_DWORD :
        F_IsAnyEqualToUnionValue := ExpectedOrActual.dwordExpectedOrActual = AnyExpectedOrActual.dwordExpectedOrActual;

    IBaseLibrary.TypeClass.TYPE_LWORD :
        F_IsAnyEqualToUnionValue := ExpectedOrActual.lwordExpectedOrActual = AnyExpectedOrActual.lwordExpectedOrActual;

    IBaseLibrary.TypeClass.TYPE_SINT :
        F_IsAnyEqualToUnionValue := ExpectedOrActual.sintExpectedOrActual = AnyExpectedOrActual.sintExpectedOrActual;

    IBaseLibrary.TypeClass.TYPE_INT :
        F_IsAnyEqualToUnionValue := ExpectedOrActual.intExpectedOrActual = AnyExpectedOrActual.intExpectedOrActual;

    IBaseLibrary.TypeClass.TYPE_DINT :
        F_IsAnyEqualToUnionValue := ExpectedOrActual.dintExpectedOrActual = AnyExpectedOrActual.dintExpectedOrActual;

    IBaseLibrary.TypeClass.TYPE_LINT :
        F_IsAnyEqualToUnionValue := ExpectedOrActual.lintExpectedOrActual = AnyExpectedOrActual.lintExpectedOrActual;

    IBaseLibrary.TypeClass.TYPE_USINT :
        F_IsAnyEqualToUnionValue := ExpectedOrActual.usintExpectedOrActual = AnyExpectedOrActual.usintExpectedOrActual;

    IBaseLibrary.TypeClass.TYPE_UINT :
        F_IsAnyEqualToUnionValue := ExpectedOrActual.uintExpectedOrActual = AnyExpectedOrActual.uintExpectedOrActual;

    IBaseLibrary.TypeClass.TYPE_UDINT :
        F_IsAnyEqualToUnionValue := ExpectedOrActual.udintExpectedOrActual = AnyExpectedOrActual.udintExpectedOrActual;

    IBaseLibrary.TypeClass.TYPE_ULINT :
        F_IsAnyEqualToUnionValue := ExpectedOrActual.ulintExpectedOrActual = AnyExpectedOrActual.ulintExpectedOrActual;

    IBaseLibrary.TypeClass.TYPE_REAL :
        F_IsAnyEqualToUnionValue := ExpectedOrActual.realExpectedOrActual = AnyExpectedOrActual.realExpectedOrActual;

    IBaseLibrary.TypeClass.TYPE_LREAL :
        F_IsAnyEqualToUnionValue := ExpectedOrActual.lrealExpectedOrActual = AnyExpectedOrActual.lrealExpectedOrActual;

    IBaseLibrary.TypeClass.TYPE_STRING :
        F_IsAnyEqualToUnionValue := ExpectedOrActual.stringExpectedOrActual = AnyExpectedOrActual.stringExpectedOrActual;

    IBaseLibrary.TypeClass.TYPE_WSTRING :
        F_IsAnyEqualToUnionValue := ExpectedOrActual.wstringExpectedOrActual = AnyExpectedOrActual.wstringExpectedOrActual;

    IBaseLibrary.TypeClass.TYPE_TIME :
        F_IsAnyEqualToUnionValue := ExpectedOrActual.timeExpectedOrActual = AnyExpectedOrActual.timeExpectedOrActual;

    IBaseLibrary.TypeClass.TYPE_DATE :
        F_IsAnyEqualToUnionValue := ExpectedOrActual.dateExpectedOrActual = AnyExpectedOrActual.dateExpectedOrActual;

    IBaseLibrary.TypeClass.TYPE_DATEANDTIME :
        F_IsAnyEqualToUnionValue := ExpectedOrActual.dateandtimeExpectedOrActual = AnyExpectedOrActual.dateandtimeExpectedOrActual;

    IBaseLibrary.TypeClass.TYPE_TIMEOFDAY :
        F_IsAnyEqualToUnionValue := ExpectedOrActual.timeofdayExpectedOrActual = AnyExpectedOrActual.timeofdayExpectedOrActual;

    IBaseLibrary.TypeClass.TYPE_POINTER :
        F_IsAnyEqualToUnionValue := FALSE;

    IBaseLibrary.TypeClass.TYPE_REFERENCE :
        F_IsAnyEqualToUnionValue := FALSE;

    IBaseLibrary.TypeClass.TYPE_SUBRANGE :
        F_IsAnyEqualToUnionValue := FALSE;

    IBaseLibrary.TypeClass.TYPE_ENUM :
        F_IsAnyEqualToUnionValue := FALSE;

    IBaseLibrary.TypeClass.TYPE_ARRAY :
        F_IsAnyEqualToUnionValue := FALSE;

    IBaseLibrary.TypeClass.TYPE_PARAMS :
        F_IsAnyEqualToUnionValue := FALSE;

    IBaseLibrary.TypeClass.TYPE_USERDEF :
        F_IsAnyEqualToUnionValue := FALSE;

    IBaseLibrary.TypeClass.TYPE_NONE :
        F_IsAnyEqualToUnionValue := FALSE;

    IBaseLibrary.TypeClass.TYPE_ANY :
        (* Even though the data input of the ExpectedOrActual is ANY, this CASE-switch will never
           enter this case, but instead the type-class that it is an instance of. So for instance,
           if the ExpectedOrActual is an instance of INT, this case-switch will enter the 
           IBaseLibrary.TypeClass.TYPE_INT case. *)
        F_IsAnyEqualToUnionValue := FALSE;

    IBaseLibrary.TypeClass.TYPE_ANYBIT :
        F_IsAnyEqualToUnionValue := FALSE;

    IBaseLibrary.TypeClass.TYPE_ANYDATE :
        F_IsAnyEqualToUnionValue := FALSE;

    IBaseLibrary.TypeClass.TYPE_ANYINT :
        F_IsAnyEqualToUnionValue := FALSE;

    IBaseLibrary.TypeClass.TYPE_ANYNUM :
        F_IsAnyEqualToUnionValue := FALSE;

    IBaseLibrary.TypeClass.TYPE_ANYREAL :
        F_IsAnyEqualToUnionValue := FALSE;

    IBaseLibrary.TypeClass.TYPE_LAZY :
        F_IsAnyEqualToUnionValue := FALSE;

    IBaseLibrary.TypeClass.TYPE_LTIME :
        F_IsAnyEqualToUnionValue := ExpectedOrActual.ltimeExpectedOrActual = AnyExpectedOrActual.ltimeExpectedOrActual;

    IBaseLibrary.TypeClass.TYPE_BITCONST :
        F_IsAnyEqualToUnionValue := FALSE;

    IBaseLibrary.TypeClass.TYPE_INTERFACE :
        F_IsAnyEqualToUnionValue := FALSE;

    ELSE
        F_IsAnyEqualToUnionValue := FALSE;
END_CASE

END_FUNCTION

// ---- POUs/FB_AssertArrayResultStatic.TcPOU
(*
    This function block is responsible for keeping track of which array-asserts that have been made.
    The reason we need to keep track of these is because if the user does the same assert twice
    (because of running a test suite over several PLC-cycles) we want to know it so we don't print several times
    (if the assert fails). An instance of an array-assert is keyed/identified with the following parameters as key:
    - Array-size (in bytes) of the expecteds
    - Datatype of the expecteds
    - Array-size (in bytes) of the actuals
    - Datatype of the actuals
    - Message (string)
    - Test instance path (string)
*)
FUNCTION_BLOCK FB_AssertArrayResultStatic
VAR
    // The total number of instances of each of the "AssertArrayResults"
    AssertArrayResults : ARRAY[1..GVL_Param_TcUnit.MaxNumberOfAssertsForEachTestSuite] OF ST_AssertArrayResult;

    // The total number of unique asserts
    TotalArrayAsserts : UINT := 0;

    // Function block to get the current task cycle
    GetCurrentTaskIndex : GETCURTASKINDEX;

    // The total number of instances of each of the "AssertArrayResults"
    AssertArrayResultInstances : ARRAY[1..GVL_Param_TcUnit.MaxNumberOfAssertsForEachTestSuite] OF ST_AssertArrayResultInstances;

    // The last PLC cycle count
    CycleCount : UDINT;

    // Only run first cycle
    FirstCycleExecuted : BOOL;
END_VAR

METHOD PRIVATE AddAssertArrayResult
VAR_INPUT
    ExpectedsSize : UDINT;
    ExpectedsTypeClass : IBaseLibrary.TypeClass;
    ActualsSize : UDINT;
    ActualsTypeClass : IBaseLibrary.TypeClass;
    Message : T_MaxString;
    TestInstancePath : T_MaxString;
END_VAR
VAR_INST
	AssertResultOverflow : BOOL := FALSE;
END_VAR
VAR
    sErrorString : T_MaxString;
END_VAR
IF TotalArrayAsserts < GVL_Param_TcUnit.MaxNumberOfAssertsForEachTestSuite THEN
	TotalArrayAsserts := TotalArrayAsserts + 1;
	AssertArrayResults[TotalArrayAsserts].ExpectedsSize := ExpectedsSize;
	AssertArrayResults[TotalArrayAsserts].ExpectedsTypeClass := ExpectedsTypeClass;
	AssertArrayResults[TotalArrayAsserts].ActualsSize := ActualsSize;
	AssertArrayResults[TotalArrayAsserts].ActualsTypeClass := ActualsTypeClass;
	AssertArrayResults[TotalArrayAsserts].Message := Message;
	AssertArrayResults[TotalArrayAsserts].TestInstancePath := TestInstancePath;
ELSE
	IF NOT AssertResultOverflow THEN
        sErrorString := CONCAT(STR1 := F_GetTestSuiteNameFromTestInstancePath(TestInstancePath := TestInstancePath),
                               STR2 := '. Max number of assertions exceeded. Check parameter MaxNumberOfAssertsForEachTestSuite.');
		GVL_TcUnit.AdsMessageQueue.WriteLog(MsgCtrlMask := ADSLOG_MSGTYPE_ERROR,
											MsgFmtStr := sErrorString,
											StrArg := '');
		AssertResultOverflow := TRUE;
	END_IF
END_IF
END_METHOD

METHOD PRIVATE CopyDetectionCountAndResetDetectionCountInThisCycle
VAR
    IteratorCounter : UINT;
END_VAR
FOR IteratorCounter := 1 TO GVL_Param_TcUnit.MaxNumberOfAssertsForEachTestSuite BY 1 DO
    AssertArrayResultInstances[IteratorCounter].DetectionCount := AssertArrayResultInstances[IteratorCounter].DetectionCountThisCycle;
    AssertArrayResultInstances[IteratorCounter].DetectionCountThisCycle := 0;
END_FOR
END_METHOD

METHOD PRIVATE CreateAssertResultInstance
VAR_INPUT
    ExpectedsSize : UDINT;
    ExpectedsTypeClass : IBaseLibrary.TypeClass;
    ActualsSize : UDINT;
    ActualsTypeClass : IBaseLibrary.TypeClass;
    Message : T_MaxString;
    TestInstancePath : T_MaxString;
END_VAR
VAR
    IteratorCounter : UINT;
END_VAR
FOR IteratorCounter := 1 TO GVL_Param_TcUnit.MaxNumberOfAssertsForEachTestSuite BY 1 DO
    IF AssertArrayResultInstances[IteratorCounter].DetectionCount = 0 AND
        AssertArrayResultInstances[IteratorCounter].DetectionCountThisCycle = 0 THEN // Find first free spot
        AssertArrayResultInstances[IteratorCounter].AssertArrayResult.ExpectedsSize := ExpectedsSize;
        AssertArrayResultInstances[IteratorCounter].AssertArrayResult.ExpectedsTypeClass := ExpectedsTypeClass;
        AssertArrayResultInstances[IteratorCounter].AssertArrayResult.ActualsSize := ActualsSize;
        AssertArrayResultInstances[IteratorCounter].AssertArrayResult.ActualsTypeClass := ActualsTypeClass;
        AssertArrayResultInstances[IteratorCounter].AssertArrayResult.Message := Message;
        AssertArrayResultInstances[IteratorCounter].AssertArrayResult.TestInstancePath := TestInstancePath;
        AssertArrayResultInstances[IteratorCounter].DetectionCountThisCycle := 1;
        EXIT;
    END_IF
END_FOR
END_METHOD

METHOD PRIVATE GetDetectionCount : UINT
VAR_INPUT
    ExpectedsSize : UDINT;
    ExpectedsTypeClass : IBaseLibrary.TypeClass;
    ActualsSize : UDINT;
    ActualsTypeClass : IBaseLibrary.TypeClass;
    Message : T_MaxString;
    TestInstancePath : T_MaxString;
END_VAR
VAR
    IteratorCounter : UINT;
END_VAR
FOR IteratorCounter := 1 TO GVL_Param_TcUnit.MaxNumberOfAssertsForEachTestSuite BY 1 DO
    IF AssertArrayResultInstances[IteratorCounter].AssertArrayResult.ExpectedsSize = ExpectedsSize AND
       AssertArrayResultInstances[IteratorCounter].AssertArrayResult.ExpectedsTypeClass = ExpectedsTypeClass AND
       AssertArrayResultInstances[IteratorCounter].AssertArrayResult.ActualsSize = ActualsSize AND
       AssertArrayResultInstances[IteratorCounter].AssertArrayResult.ActualsTypeClass = ActualsTypeClass AND
       AssertArrayResultInstances[IteratorCounter].AssertArrayResult.Message = Message AND
       AssertArrayResultInstances[IteratorCounter].AssertArrayResult.TestInstancePath = TestInstancePath THEN
        GetDetectionCount := AssertArrayResultInstances[IteratorCounter].DetectionCount;
    END_IF
END_FOR
END_METHOD

METHOD PRIVATE GetDetectionCountThisCycle : UINT
VAR_INPUT
    ExpectedsSize : UDINT;
    ExpectedsTypeClass : IBaseLibrary.TypeClass;
    ActualsSize : UDINT;
    ActualsTypeClass : IBaseLibrary.TypeClass;
    Message : T_MaxString;
    TestInstancePath : T_MaxString;
END_VAR
VAR
    IteratorCounter : UINT;
END_VAR
FOR IteratorCounter := 1 TO GVL_Param_TcUnit.MaxNumberOfAssertsForEachTestSuite BY 1 DO
    IF AssertArrayResultInstances[IteratorCounter].AssertArrayResult.ExpectedsSize = ExpectedsSize AND
       AssertArrayResultInstances[IteratorCounter].AssertArrayResult.ExpectedsTypeClass = ExpectedsTypeClass AND
       AssertArrayResultInstances[IteratorCounter].AssertArrayResult.ActualsSize = ActualsSize AND
       AssertArrayResultInstances[IteratorCounter].AssertArrayResult.ActualsTypeClass = ActualsTypeClass AND
       AssertArrayResultInstances[IteratorCounter].AssertArrayResult.Message = Message AND
       AssertArrayResultInstances[IteratorCounter].AssertArrayResult.TestInstancePath = TestInstancePath THEN

        GetDetectionCountThisCycle := AssertArrayResultInstances[IteratorCounter].DetectionCountThisCycle;
    END_IF
END_FOR
END_METHOD

METHOD INTERNAL GetNumberOfArrayAssertsForTest : UINT
VAR_INPUT
    CompleteTestInstancePath : T_MaxString;
END_VAR
VAR
    Counter : UINT;
    NumberOfArrayAsserts : UINT := 0;
END_VAR
IF TotalArrayAsserts > 0 THEN
    FOR Counter := 1 TO TotalArrayAsserts BY 1 DO
        IF AssertArrayResults[Counter].TestInstancePath = CompleteTestInstancePath THEN
            NumberOfArrayAsserts := NumberOfArrayAsserts + 1;
        END_IF
    END_FOR
END_IF

GetNumberOfArrayAssertsForTest := NumberOfArrayAsserts;
END_METHOD

(*
    This method is called in every assert and returns whether this particular assert has already been called.
    The reason one would like to know whether this assert has already been reported or not is to not report it several
    times to any logging service. Because a test-suite can consist of several tests, and certain tests can require the
    test to run over several cycles it means that certain asserts could be called several times and thus we need to
    keep track of which asserts we've already reported. The user of the framework should not need to care for any of
    this and he/she should be able to call the asserts in any way they find suitable.

    To know what assert this is we need to check for the total combination of:
    - Test message
    - Test instance path
    - Expecteds size (in bytes)
    - Actuals size (in bytes)
    - Expecteds datatype
    - Actuals datatype
    Theoretically we can have a situation where a test has three different asserts, each and one with the same test
    message/test instance path/actuals size&datatype/expecteds size&datatype but called within the same or different
    cycles. In order for us to handle all situations we need a simple algorithm that works according to:
    - Keep track of how many instances the combination of test message/test instance path/expecteds size&datatype/
      actuals size&datatype we have. So for example, if we have called
      Assert(Exp := [5,4,3], Act := [5,4,3], 'Hello there', 'PRG.InstanceTestSuite.Test')
      two times in one cycle, we have two instances of that combination. This is done according to:
    - Iterate all existing reports.
      - If we have a new PLC-cycle, set the current detection-count to zero.
      - If new report does not match in any of the above fields, create it (together with current PLC-cycle).
        Also store the information that we have one instance of this combination and +1 on the detection-count.
      - If new report matches in all of the above, +1 in the detection-count. If this detection-count is larger than
        the stored detection-count for this combination, create a new report and add +1 to the storage of
        the detection-count.
*)
METHOD INTERNAL ReportResult
VAR_INPUT
    ExpectedsSize : UDINT;
    ExpectedsTypeClass : IBaseLibrary.TypeClass;
    ActualsSize : UDINT;
    ActualsTypeClass : IBaseLibrary.TypeClass;
    Message : T_MaxString;
    TestInstancePath : T_MaxString;
END_VAR
VAR_OUTPUT
    AlreadyReported : BOOL := FALSE;
END_VAR
VAR
    LocationIndex : UINT;
    DataTypesNotEquals : BOOL;
    DataSizeNotEquals : BOOL;
    DataContentNotEquals : BOOL;
    CurrentCycleCount : UDINT;
    IteratorCounter : UINT;
    DetectionCountTemp : UINT := 0;
    FoundOne : BOOL;
    AdditionalIdenticalAssert : BOOL;
END_VAR
IF NOT FirstCycleExecuted THEN
    GetCurrentTaskIndex();
    FirstCycleExecuted := TRUE;
END_IF

CurrentCycleCount := TwinCAT_SystemInfoVarList._TaskInfo[GetCurrentTaskIndex.index].CycleCount;
(* Is current cycle the same as the last call to this method?
   If not, reset the detection count *)
IF CurrentCycleCount <> CycleCount THEN
    CopyDetectionCountAndResetDetectionCountInThisCycle();
END_IF

FOR IteratorCounter := 1 TO TotalArrayAsserts BY 1 DO
    IF AssertArrayResultInstances[IteratorCounter].AssertArrayResult.ExpectedsSize = ExpectedsSize AND
        AssertArrayResultInstances[IteratorCounter].AssertArrayResult.ExpectedsTypeClass = ExpectedsTypeClass AND
        AssertArrayResultInstances[IteratorCounter].AssertArrayResult.ActualsSize = ActualsSize AND
        AssertArrayResultInstances[IteratorCounter].AssertArrayResult.ActualsTypeClass = ActualsTypeClass AND
        AssertArrayResultInstances[IteratorCounter].AssertArrayResult.Message = Message AND
        AssertArrayResultInstances[IteratorCounter].AssertArrayResult.TestInstancePath = TestInstancePath THEN
        AssertArrayResultInstances[IteratorCounter].DetectionCountThisCycle :=
            AssertArrayResultInstances[IteratorCounter].DetectionCountThisCycle + 1;
            FoundOne := TRUE;
        IF AssertArrayResultInstances[IteratorCounter].DetectionCountThisCycle >
                AssertArrayResultInstances[IteratorCounter].DetectionCount THEN // This assert is new
                AdditionalIdenticalAssert := TRUE;
        END_IF
        EXIT;
    END_IF
END_FOR

// If not found anything, create the first
IF NOT FoundOne THEN
    // No existing match found, create a new entry
    AddAssertArrayResult(ExpectedsSize := ExpectedsSize,
                         ExpectedsTypeClass := ExpectedsTypeClass,
                         ActualsSize := ActualsSize,
                         ActualsTypeClass := ActualsTypeClass,
                         Message := Message,
                         TestInstancePath := TestInstancePath);
    CreateAssertResultInstance(ExpectedsSize := ExpectedsSize,
                               ExpectedsTypeClass := ExpectedsTypeClass,
                               ActualsSize := ActualsSize,
                               ActualsTypeClass := ActualsTypeClass,
                               Message := Message,
                               TestInstancePath := TestInstancePath);
// An additional instance of this assert needs to be created
ELSIF AdditionalIdenticalAssert THEN
    AddAssertArrayResult(ExpectedsSize := ExpectedsSize,
                         ExpectedsTypeClass := ExpectedsTypeClass,
                         ActualsSize := ActualsSize,
                         ActualsTypeClass := ActualsTypeClass,
                         Message := Message,
                         TestInstancePath := TestInstancePath);
// In all other cases, this assert has already been reported, we don't need to do anything
ELSE
    AlreadyReported := TRUE;
END_IF

// Update the cycle count
CycleCount := TwinCAT_SystemInfoVarList._TaskInfo[GetCurrentTaskIndex.index].CycleCount;
END_METHOD

END_FUNCTION_BLOCK

// ---- POUs/FB_AdsAssertMessageFormatter.TcPOU
(*
    This function block is responsible for printing the results of the assertions using the built-in
    ADSLOGSTR functionality provided by the Tc2_System library. This sends the result using ADS, which
    is consumed by the error list of Visual Studio.
*)
FUNCTION_BLOCK FB_AdsAssertMessageFormatter IMPLEMENTS I_AssertMessageFormatter

METHOD PUBLIC LogAssertFailure
VAR_INPUT
    Expected : T_MaxString;
    Actual : T_MaxString;
    Message : T_MaxString;
    TestInstancePath : T_MaxString;
END_VAR
VAR
    AdjustAssertFailureMessageToMaxAllowedLength : FB_AdjustAssertFailureMessageToMaxAllowedLength;
    TestInstancePathCleaned : T_MaxString;
    TestInstancePathFinal : T_MaxString;
    ReturnValue : DINT;
    TestInstancePathProcessed : T_MaxString;
    MessagePart2 : T_MaxString;
    MessagePart3 : T_MaxString;
    MessagePart4 : T_MaxString;
    MessageProcessed : T_MaxString;
    Length2 : INT;
    Length3 : INT;
    Length4 : INT;
    LengthTotal : INT;
END_VAR
VAR CONSTANT
    MESSAGE_FORMATTED_STRING_MAX_NUMBER_OF_CHARACTERS : INT := 252; // The maximum printed text length is 250. The '%s' placeholder will be replaced, therefore the limit to use in the check is 252.
    ACTEXP_MAX_NUMBER_OF_CHARACTERS : INT := 250;
    TOO_LONG : STRING := '...too long';
END_VAR
TestInstancePathCleaned := F_RemoveInstancePathAndProjectNameFromTestInstancePath(TestInstancePath);
TestInstancePathFinal := CONCAT(STR1 := 'FAILED TEST $'',
                                STR2 := TestInstancePathCleaned);
TestInstancePathFinal := CONCAT(STR1 := TestInstancePathFinal,
                                STR2 := '$'');

MessagePart2 := CONCAT(STR1 := 'EXP: ',
                       STR2 := Expected);
MessagePart3 := CONCAT(STR1 := 'ACT: ',
                       STR2 := Actual);
IF LEN(STR := Message) > 0 THEN
    MessagePart4 := ', MSG: %s';
    Length4 := LEN(STR := MessagePart4)
             + LEN(STR := Message);
END_IF

IF (GVL_Param_TcUnit.MultipleLinesPerAssertionMessage) THEN
    Length2 := LEN(MessagePart2);
    IF (Length2 > ACTEXP_MAX_NUMBER_OF_CHARACTERS) THEN
        MessagePart2 := LEFT(STR := MessagePart2,
                             SIZE := ACTEXP_MAX_NUMBER_OF_CHARACTERS - LEN(STR := TOO_LONG));
        MessagePart2 := CONCAT (STR1 := MessagePart2,
                                STR2 := TOO_LONG);
        Length2 := LEN(MessagePart2);
    END_IF
    
    Length3 := LEN(MessagePart3);
    IF (Length3 > ACTEXP_MAX_NUMBER_OF_CHARACTERS) THEN
        MessagePart3 := LEFT(STR := MessagePart3,
                             SIZE := ACTEXP_MAX_NUMBER_OF_CHARACTERS - LEN(STR := TOO_LONG));
        MessagePart3 := CONCAT (STR1 := MessagePart3,
                                STR2 := TOO_LONG);
        Length3 := LEN(MessagePart3);
    END_IF

    LengthTotal := LEN(TestInstancePathFinal) + 2 + Length2 + 2 + Length3 + Length4;
END_IF

IF (LengthTotal <= MESSAGE_FORMATTED_STRING_MAX_NUMBER_OF_CHARACTERS) THEN
    // If the message must be printed on a single line ("multiple lines" disabled), then LengthTotal is not calculated, so this path is executed.
    TestInstancePathFinal := CONCAT(STR1 := TestInstancePathFinal,
                                    STR2 := ', ');
    TestInstancePathFinal := CONCAT(STR1 := TestInstancePathFinal,
                                    STR2 := MessagePart2);
    
    TestInstancePathFinal := CONCAT(STR1 := TestInstancePathFinal,
                                    STR2 := ', ');
    TestInstancePathFinal := CONCAT(STR1 := TestInstancePathFinal,
                                    STR2 := MessagePart3);
    
    IF Length4 > 0 THEN
        TestInstancePathFinal := CONCAT(STR1 := TestInstancePathFinal,
                                        STR2 := MessagePart4);
    END_IF
    
    AdjustAssertFailureMessageToMaxAllowedLength(TestInstancePath := TestInstancePathFinal,
                                                 TestMessage := Message,
                                                 TestInstancePathProcessed => TestInstancePathProcessed,
                                                 TestMessageProcessed => MessageProcessed);
    
    GVL_TcUnit.AdsMessageQueue.WriteLog(MsgCtrlMask := ADSLOG_MSGTYPE_ERROR,
                                        MsgFmtStr := TestInstancePathProcessed,
                                        StrArg := MessageProcessed);
    
// ELSE: print multiple lines
ELSIF (LEN(TestInstancePathFinal) + 2 + Length2 + 2 + Length3 <= MESSAGE_FORMATTED_STRING_MAX_NUMBER_OF_CHARACTERS) THEN
    // A message exists, because the text with message does not fit in one line, but it fits without the message. Print only the message in a separate line.
    TestInstancePathFinal := CONCAT(STR1 := TestInstancePathFinal,
                                    STR2 := ', ');
    TestInstancePathFinal := CONCAT(STR1 := TestInstancePathFinal,
                                    STR2 := MessagePart2);
    
    TestInstancePathFinal := CONCAT(STR1 := TestInstancePathFinal,
                                    STR2 := ', ');
    TestInstancePathFinal := CONCAT(STR1 := TestInstancePathFinal,
                                    STR2 := MessagePart3);
    
    AdjustAssertFailureMessageToMaxAllowedLength(TestInstancePath := TestInstancePathFinal,
                                                 TestMessage := '',
                                                 TestInstancePathProcessed => TestInstancePathProcessed,
                                                 TestMessageProcessed => MessageProcessed);
    
    GVL_TcUnit.AdsMessageQueue.WriteLog(MsgCtrlMask := ADSLOG_MSGTYPE_ERROR,
                                        MsgFmtStr := TestInstancePathProcessed,
                                        StrArg := MessageProcessed);
    
    // MessagePart4 (MSG)
    AdjustAssertFailureMessageToMaxAllowedLength(TestInstancePath := '_ MSG: %s',
                                                 TestMessage := Message,
                                                 TestInstancePathProcessed => TestInstancePathProcessed,
                                                 TestMessageProcessed => MessageProcessed);
    
    GVL_TcUnit.AdsMessageQueue.WriteLog(MsgCtrlMask := ADSLOG_MSGTYPE_ERROR,
                                        MsgFmtStr := TestInstancePathProcessed,
                                        StrArg := MessageProcessed);
    
ELSIF (2 + Length2 + 2 + Length3 <= ACTEXP_MAX_NUMBER_OF_CHARACTERS) THEN
    // Text without message does not fit in one line. EXP and ACT fit in one line, therefore print them together in 2nd line. Print message (if existing) in 3rd line.
    AdjustAssertFailureMessageToMaxAllowedLength(TestInstancePath := TestInstancePathFinal,
                                                 TestMessage := '',
                                                 TestInstancePathProcessed => TestInstancePathProcessed,
                                                 TestMessageProcessed => MessageProcessed);
    
    GVL_TcUnit.AdsMessageQueue.WriteLog(MsgCtrlMask := ADSLOG_MSGTYPE_ERROR,
                                        MsgFmtStr := TestInstancePathProcessed,
                                        StrArg := MessageProcessed);
    
    // MessagePart2 (EXP) + MessagePart3 (ACT)
    MessagePart2 := CONCAT (STR1 := '_ ',
                            STR2 := MessagePart2);
    MessagePart2 := CONCAT (STR1 := MessagePart2,
                            STR2 := ', ');
    MessagePart2 := CONCAT (STR1 := MessagePart2,
                            STR2 := MessagePart3);
    
    AdjustAssertFailureMessageToMaxAllowedLength(TestInstancePath := MessagePart2,
                                                 TestMessage := '',
                                                 TestInstancePathProcessed => TestInstancePathProcessed,
                                                 TestMessageProcessed => MessageProcessed);
    
    GVL_TcUnit.AdsMessageQueue.WriteLog(MsgCtrlMask := ADSLOG_MSGTYPE_ERROR,
                                        MsgFmtStr := TestInstancePathProcessed,
                                        StrArg := MessageProcessed);
    
    // MessagePart4 (MSG)
    IF Length4 > 0 THEN
        AdjustAssertFailureMessageToMaxAllowedLength(TestInstancePath := '_ MSG: %s',
                                                     TestMessage := Message,
                                                     TestInstancePathProcessed => TestInstancePathProcessed,
                                                     TestMessageProcessed => MessageProcessed);
        
        GVL_TcUnit.AdsMessageQueue.WriteLog(MsgCtrlMask := ADSLOG_MSGTYPE_ERROR,
                                            MsgFmtStr := TestInstancePathProcessed,
                                            StrArg := MessageProcessed);
    END_IF
ELSE
    // print every item in a separate line.
    AdjustAssertFailureMessageToMaxAllowedLength(TestInstancePath := TestInstancePathFinal,
                                                 TestMessage := '',
                                                 TestInstancePathProcessed => TestInstancePathProcessed,
                                                 TestMessageProcessed => MessageProcessed);
    
    GVL_TcUnit.AdsMessageQueue.WriteLog(MsgCtrlMask := ADSLOG_MSGTYPE_ERROR,
                                        MsgFmtStr := TestInstancePathProcessed,
                                        StrArg := MessageProcessed);
    
    // MessagePart2 (EXP)
    MessagePart2 := CONCAT (STR1 := '_ ',
                            STR2 := MessagePart2);

    AdjustAssertFailureMessageToMaxAllowedLength(TestInstancePath := MessagePart2,
                                                 TestMessage := '',
                                                 TestInstancePathProcessed => TestInstancePathProcessed,
                                                 TestMessageProcessed => MessageProcessed);
    
    GVL_TcUnit.AdsMessageQueue.WriteLog(MsgCtrlMask := ADSLOG_MSGTYPE_ERROR,
                                        MsgFmtStr := TestInstancePathProcessed,
                                        StrArg := MessageProcessed);
    
    // MessagePart3 (ACT)
    MessagePart3 := CONCAT (STR1 := '_ ',
                            STR2 := MessagePart3);
    
    AdjustAssertFailureMessageToMaxAllowedLength(TestInstancePath := MessagePart3,
                                                 TestMessage := '',
                                                 TestInstancePathProcessed => TestInstancePathProcessed,
                                                 TestMessageProcessed => MessageProcessed);
    
    GVL_TcUnit.AdsMessageQueue.WriteLog(MsgCtrlMask := ADSLOG_MSGTYPE_ERROR,
                                        MsgFmtStr := TestInstancePathProcessed,
                                        StrArg := MessageProcessed);
    
    // MessagePart4 (MSG)
    IF Length4 > 0 THEN
        AdjustAssertFailureMessageToMaxAllowedLength(TestInstancePath := '_ MSG: %s',
                                                     TestMessage := Message,
                                                     TestInstancePathProcessed => TestInstancePathProcessed,
                                                     TestMessageProcessed => MessageProcessed);
        
        GVL_TcUnit.AdsMessageQueue.WriteLog(MsgCtrlMask := ADSLOG_MSGTYPE_ERROR,
                                            MsgFmtStr := TestInstancePathProcessed,
                                            StrArg := MessageProcessed);
    END_IF
END_IF
END_METHOD

END_FUNCTION_BLOCK

// ---- POUs/FB_AdjustAssertFailureMessageToMaxAllowedLength.TcPOU
(*
    This function block is responsible for making sure that the asserted test instance path and test message are not
    loo long. The total printed message can not be more than 250 characters long.
*)
FUNCTION_BLOCK FB_AdjustAssertFailureMessageToMaxAllowedLength
VAR_INPUT
    TestInstancePath : T_MaxString;
    TestMessage : T_MaxString;
END_VAR
VAR_OUTPUT
    TestInstancePathProcessed : T_MaxString;
    TestMessageProcessed : T_MaxString;
END_VAR
VAR_TEMP
    TestInstancePathLen : INT;
    TestMessageLen : INT;
    TestInstancePathTemporary : T_MaxString;
END_VAR
VAR CONSTANT
    MESSAGE_FORMATTED_STRING_MAX_NUMBER_OF_CHARACTERS : INT := 252; // The maximum printed text length is 250. The '%s' placeholder will be replaced, therefore the limit to use in the check is 252.
    TEST_NAME_TOO_LONG : STRING := '...TestName too long';
    TEST_MESSAGE_TOO_LONG : STRING := '...TestMsg too long';
END_VAR

// Check if any of the two strings are too long (or the combination of them)

TestInstancePathLen := LEN(STR := TestInstancePath);
TestMessageLen      := LEN(STR := TestMessage);

